  gc_DbmTranslation_fr_Text2200 : WSTRING(29) := "Activate Measuring Mast (A21)";
  gc_DbmTranslation_fr_Text2201 : WSTRING(76) := "Button for the calibration of min position mast measure encodeur  is pressed";
  gc_DbmTranslation_fr_Text2202 : WSTRING(76) := "Button for the calibration of max position mast measure encodeur  is pressed";
  gc_DbmTranslation_fr_Text2203 : WSTRING(58) := "Button for save min and max value of encodeur mast measure";
  gc_DbmTranslation_fr_Text2204 : WSTRING(60) := "Raz distance translation traveled with mast measure unfolded";
  gc_DbmTranslation_fr_Text2205 : WSTRING(13) := "Serial Number";
  gc_DbmTranslation_fr_Text2206 : WSTRING(18) := "BP Basket Validate";
  gc_DbmTranslation_fr_Text2207 : WSTRING(19) := "Key Filter Overload";
  gc_DbmTranslation_fr_Text2208 : WSTRING(13) := "Key Next Mode";
  gc_DbmTranslation_fr_Text2209 : WSTRING(13) := "Key Prev Mode";
  gc_DbmTranslation_fr_Text2210 : WSTRING(17) := "Key Signal Danger";
  gc_DbmTranslation_fr_Text2211 : WSTRING(18) := "Key Flash Light ON";
  gc_DbmTranslation_fr_Text2212 : WSTRING(18) := "Key Calib Mast Min";
  gc_DbmTranslation_fr_Text2213 : WSTRING(18) := "Key Calib Mast Max";
  gc_DbmTranslation_fr_Text2214 : WSTRING(17) := "KeyCalibMastValid";
  gc_DbmTranslation_fr_Text2215 : WSTRING(24) := "Key Generator Activation";
  gc_DbmTranslation_fr_Text2216 : WSTRING(31) := "Bypass pressure threshold alarm";
  gc_DbmTranslation_fr_Text2217 : WSTRING(66) := "DM_TELESCOPE_SENSOR_FAULT - Telescope In torlerance with inductive";
  gc_DbmTranslation_fr_Text2218 : WSTRING(78) := "DM_TELESCOPE_SENSOR_FAULT - Telescope torlerance when no movement is solicited";
  gc_DbmTranslation_fr_Text2219 : WSTRING(68) := "DM_TELESCOPE_SENSOR_FAULT - Telescope torlerance beetween 2 Channels";
  gc_DbmTranslation_fr_Text2220 : WSTRING(64) := "DM__INC_ALTERNATOR_CHARGE_FAULT - max treshold alternator regime";
  gc_DbmTranslation_fr_Text2221 : WSTRING(62) := "DM__INC_ALTERNATOR_CHARGE_FAULT - min treshold battery voltage";
  gc_DbmTranslation_fr_Text2222 : WSTRING(108) := "DM_C1_OUT_OF_RANGE_JOY_DELTA_ARM_48XS - min alarm value of joytick delta arm in % according batterie voltage";
  gc_DbmTranslation_fr_Text2223 : WSTRING(108) := "DM_C1_OUT_OF_RANGE_JOY_DELTA_ARM_48XS - max alarm value of joytick delta arm in % according batterie voltage";
  gc_DbmTranslation_fr_Text2224 : WSTRING(108) := "DM_C1_OUT_OF_RANGE_JOY_ARROW_ARM_48XS - min alarm value of joytick arrow arm in % according batterie voltage";
  gc_DbmTranslation_fr_Text2225 : WSTRING(108) := "DM_C1_OUT_OF_RANGE_JOY_ARROW_ARM_48XS - max alarm value of joytick arrow arm in % according batterie voltage";
  gc_DbmTranslation_fr_Text2226 : WSTRING(116) := "DM_C1_OUT_OF_RANGE_JOY_TELESCOPE_ARM_48XS - min alarm value of joytick telescope arm in % according batterie voltage";
  gc_DbmTranslation_fr_Text2227 : WSTRING(116) := "DM_C1_OUT_OF_RANGE_JOY_TELESCOPE_ARM_48XS - max alarm value of joytick telescope arm in % according batterie voltage";
  gc_DbmTranslation_fr_Text2228 : WSTRING(123) := "DM_C1_OUT_OF_RANGE_JOY_ROT_TURRET_ARM_48XS - min alarm value of joytick rotation turret arm in % according batterie voltage";
  gc_DbmTranslation_fr_Text2229 : WSTRING(123) := "DM_C1_OUT_OF_RANGE_JOY_ROT_TURRET_ARM_48XS - max alarm value of joytick rotation turret arm in % according batterie voltage";
  gc_DbmTranslation_fr_Text2230 : WSTRING(120) := "DM_C1_OUT_OF_RANGE_JOY_ADVANCEMENT_48XS - min alarm value of joytick rotation turret arm in % according batterie voltage";
  gc_DbmTranslation_fr_Text2231 : WSTRING(120) := "DM_C1_OUT_OF_RANGE_JOY_ADVANCEMENT_48XS - max alarm value of joytick rotation turret arm in % according batterie voltage";
  gc_DbmTranslation_fr_Text2232 : WSTRING(17) := "Time Bypass Fault";
  gc_DbmTranslation_fr_Text2233 : WSTRING(26) := "Timer for the Bypass fault";
  gc_DbmTranslation_fr_Text2234 : WSTRING(42) := "Inconsistency Nc No logical frame rotation";
  gc_DbmTranslation_fr_Text2235 : WSTRING(65) := "internal error , inconsistency between two channels and can error";
  gc_DbmTranslation_fr_Text2236 : WSTRING(37) := "Fault of Ev park brake axle osccilant";
  gc_DbmTranslation_fr_Text2237 : WSTRING(32) := "Fault of Ev park brake axle fixe";
  gc_DbmTranslation_fr_Text2238 : WSTRING(40) := "Fault of Ev service brake axle osccilant";
  gc_DbmTranslation_fr_Text2239 : WSTRING(35) := "Fault of Ev service brake axle fixe";
  gc_DbmTranslation_fr_Text2240 : WSTRING(30) := "Fault of Ev serice brake track";
  gc_DbmTranslation_fr_Text2241 : WSTRING(27) := "RM com can radio loss by C0";
  gc_DbmTranslation_fr_Text2242 : WSTRING(33) := "Ev 2nd Park Brake Axle Fixe Fault";
  gc_DbmTranslation_fr_Text2243 : WSTRING(33) := "Ev 2nd Park Brake Axle Osci Fault";
  gc_DbmTranslation_fr_Text2244 : WSTRING(0) := "";
  gc_DbmTranslation_fr_Text2245 : WSTRING(0) := "";
  gc_DbmTranslation_fr_Text2246 : WSTRING(0) := "";
  gc_DbmTranslation_fr_Text2247 : WSTRING(0) := "";
  gc_DbmTranslation_fr_Text2248 : WSTRING(0) := "";
  gc_DbmTranslation_fr_Text2249 : WSTRING(0) := "";
  gc_DbmTranslation_fr_Text2250 : WSTRING(0) := "";
  gc_DbmTranslation_fr_Text2251 : WSTRING(0) := "";
  gc_DbmTranslation_fr_Text2252 : WSTRING(0) := "";
  gc_DbmTranslation_fr_Text2253 : WSTRING(0) := "";
  gc_DbmTranslation_fr_Text2254 : WSTRING(0) := "";
  gc_DbmTranslation_fr_Text2255 : WSTRING(0) := "";
  gc_DbmTranslation_fr_Text2256 : WSTRING(0) := "";
  gc_DbmTranslation_fr_Text2257 : WSTRING(28) := "Additionnal Performance Func";
  gc_DbmTranslation_fr_Text2258 : WSTRING(21) := "Slope Case Less 2 Deg";
  gc_DbmTranslation_fr_Text2259 : WSTRING(21) := "Slope Case Less 4 Deg";
  gc_DbmTranslation_fr_Text2260 : WSTRING(21) := "Slope Case Less 6 Deg";
  gc_DbmTranslation_fr_Text2261 : WSTRING(23) := "Slope Case Higher 6 Deg";
  gc_DbmTranslation_fr_Text2262 : WSTRING(26) := "Turret In Speed Zone 2 Deg";
  gc_DbmTranslation_fr_Text2263 : WSTRING(26) := "Turret In Speed Zone 4 Deg";
  gc_DbmTranslation_fr_Text2264 : WSTRING(37) := "Turret In Speed Zone 2 Deg For Basket";
  gc_DbmTranslation_fr_Text2265 : WSTRING(21) := "Selected control post";
  gc_DbmTranslation_fr_Text2266 : WSTRING(23) := "Mast sensor position UP";
  gc_DbmTranslation_fr_Text2267 : WSTRING(40) := "Hydraulic valve uin down position sensor";
  gc_DbmTranslation_fr_Text2268 : WSTRING(28) := "Measuring mast sensor folded";
  gc_DbmTranslation_fr_Text2269 : WSTRING(35) := "Presence of sensor plate on machine";
  gc_DbmTranslation_fr_Text2270 : WSTRING(51) := "Recovery reduction ratio for the battery protection";
  gc_DbmTranslation_fr_Text2271 : WSTRING(21) := "Variable debug Neotec";
  gc_DbmTranslation_fr_Text2272 : WSTRING(21) := "Variable debug Neotec";
  gc_DbmTranslation_fr_Text2273 : WSTRING(21) := "Variable debug Neotec";
  gc_DbmTranslation_fr_Text2274 : WSTRING(21) := "Variable debug Neotec";
  gc_DbmTranslation_fr_Text2275 : WSTRING(21) := "Variable debug Neotec";
  gc_DbmTranslation_fr_Text2276 : WSTRING(21) := "Variable debug Neotec";
  gc_DbmTranslation_fr_Text2277 : WSTRING(21) := "Variable debug Neotec";
  gc_DbmTranslation_fr_Text2278 : WSTRING(21) := "Variable debug Neotec";
  gc_DbmTranslation_fr_Text2279 : WSTRING(21) := "Variable debug Neotec";
  gc_DbmTranslation_fr_Text2280 : WSTRING(21) := "Variable debug Neotec";
  gc_DbmTranslation_fr_Text2281 : WSTRING(21) := "Variable debug Neotec";
  gc_DbmTranslation_fr_Text2282 : WSTRING(21) := "Variable debug Neotec";
  gc_DbmTranslation_fr_Text2283 : WSTRING(21) := "Variable debug Neotec";
  gc_DbmTranslation_fr_Text2284 : WSTRING(21) := "Variable debug Neotec";
  gc_DbmTranslation_fr_Text2285 : WSTRING(21) := "Variable debug Neotec";
  gc_DbmTranslation_fr_Text2286 : WSTRING(21) := "Variable debug Neotec";
  gc_DbmTranslation_fr_Text2287 : WSTRING(21) := "Variable debug Neotec";
  gc_DbmTranslation_fr_Text2288 : WSTRING(21) := "Variable debug Neotec";
  gc_DbmTranslation_fr_Text2289 : WSTRING(21) := "Variable debug Neotec";
  gc_DbmTranslation_fr_Text2290 : WSTRING(21) := "Variable debug Neotec";
  gc_DbmTranslation_fr_Text2291 : WSTRING(21) := "Variable debug Neotec";
  gc_DbmTranslation_fr_Text2292 : WSTRING(21) := "Variable debug Neotec";
  gc_DbmTranslation_fr_Text2293 : WSTRING(21) := "Variable debug Neotec";
  gc_DbmTranslation_fr_Text2294 : WSTRING(21) := "Variable debug Neotec";
  gc_DbmTranslation_fr_Text2295 : WSTRING(21) := "Variable debug Neotec";
  gc_DbmTranslation_fr_Text2296 : WSTRING(21) := "Variable debug Neotec";
  gc_DbmTranslation_fr_Text2297 : WSTRING(21) := "Variable debug Neotec";
  gc_DbmTranslation_fr_Text2298 : WSTRING(21) := "Variable debug Neotec";
  gc_DbmTranslation_fr_Text2299 : WSTRING(21) := "Variable debug Neotec";
  gc_DbmTranslation_fr_Text2300 : WSTRING(21) := "Variable debug Neotec";
  gc_DbmTranslation_fr_Text2301 : WSTRING(21) := "Variable debug Neotec";
  gc_DbmTranslation_fr_Text2302 : WSTRING(21) := "Variable debug Neotec";
  gc_DbmTranslation_fr_Text2303 : WSTRING(21) := "Variable debug Neotec";
  gc_DbmTranslation_fr_Text2304 : WSTRING(21) := "Variable debug Neotec";
  gc_DbmTranslation_fr_Text2305 : WSTRING(21) := "Variable debug Neotec";
  gc_DbmTranslation_fr_Text2306 : WSTRING(21) := "Variable debug Neotec";
  gc_DbmTranslation_fr_Text2307 : WSTRING(21) := "Variable debug Neotec";
  gc_DbmTranslation_fr_Text2308 : WSTRING(21) := "Variable debug Neotec";
  gc_DbmTranslation_fr_Text2309 : WSTRING(21) := "Variable debug Neotec";
  gc_DbmTranslation_fr_Text2310 : WSTRING(21) := "Variable debug Neotec";
  gc_DbmTranslation_fr_Text2311 : WSTRING(64) := "Mesure de la température du liquide de refroidissement du moteur";
  gc_DbmTranslation_fr_Text2312 : WSTRING(58) := "Pression mesuré dans le système de lubrification du moteur";
  gc_DbmTranslation_fr_Text2313 : WSTRING(34) := "Vitesse actuelle du moteur calculé";
  gc_DbmTranslation_fr_Text2314 : WSTRING(56) := "Courant de l'alternateur principale du moteur thermique ";
  gc_DbmTranslation_fr_Text2315 : WSTRING(56) := "Etat du moteur : Motor stop, pre-start, Wram-Up,Starting";
  gc_DbmTranslation_fr_Text2316 : WSTRING(40) := "Tension mesuré aux bornes de la batterie";
  gc_DbmTranslation_fr_Text2317 : WSTRING(33) := "Commande de la vietesse du moteur";
  gc_DbmTranslation_fr_Text2318 : WSTRING(30) := "Override Control Mode (SPN695)";
  gc_DbmTranslation_fr_Text2319 : WSTRING(18) := "High pressure Oil ";
  gc_DbmTranslation_fr_Text2320 : WSTRING(14) := "Warmin gActive";
  gc_DbmTranslation_fr_Text2321 : WSTRING(10) := "Stop Motor";
  gc_DbmTranslation_fr_Text2322 : WSTRING(27) := "Regeneration SOC at maximum";
  gc_DbmTranslation_fr_Text2323 : WSTRING(61) := "Threshold maximum to autorize regeneration (Threshold of SOC)";
  gc_DbmTranslation_fr_Text2324 : WSTRING(42) := "Hysteresis for regeneration of SOC maximum";
  gc_DbmTranslation_fr_Text2325 : WSTRING(57) := "Number of time to refuse reloading from generator (Alarm)";
  gc_DbmTranslation_fr_Text2326 : WSTRING(61) := "Number of time to refuse reloading from generator (forbidden)";
  gc_DbmTranslation_fr_Text2327 : WSTRING(23) := "RPM motor maximum value";
  gc_DbmTranslation_fr_Text2328 : WSTRING(23) := "RPM motor minimum value";
  gc_DbmTranslation_fr_Text2329 : WSTRING(27) := "RPM for a movement with PVG";
  gc_DbmTranslation_fr_Text2330 : WSTRING(27) := "RPM for a movement with TOR";
  gc_DbmTranslation_fr_Text2331 : WSTRING(30) := "Hydraulic oil cold temperature";
  gc_DbmTranslation_fr_Text2332 : WSTRING(42) := "Capacity of the battery in ampere per hour";
  gc_DbmTranslation_fr_Text2333 : WSTRING(53) := "Number of element for the remaining regeneration time";
  gc_DbmTranslation_fr_Text2334 : WSTRING(61) := "Number of times the alarm regeneration threshold was exceeded";
  gc_DbmTranslation_fr_Text2335 : WSTRING(89) := "Number of times we exceeded the threshold of regeneration forbidden of the electric motor";
  gc_DbmTranslation_fr_Text2336 : WSTRING(25) := "Cold Oil Tank Temperature";
  gc_DbmTranslation_fr_Text2337 : WSTRING(30) := "Rpm Movements on Electric Mode";
  gc_DbmTranslation_fr_Text2338 : WSTRING(37) := "Rpm Translation on Rail Electric Mode";
  gc_DbmTranslation_fr_Text2339 : WSTRING(24) := "Rpm Oil Tank Temperature";
  gc_DbmTranslation_fr_Text2340 : WSTRING(18) := "Rpm Electric motor";
  gc_DbmTranslation_fr_Text2341 : WSTRING(12) := "Generator ON";
  gc_DbmTranslation_fr_Text2342 : WSTRING(23) := "Automatic mode activate";
  gc_DbmTranslation_fr_Text2343 : WSTRING(21) := "Silence mode activate";
  gc_DbmTranslation_fr_Text2344 : WSTRING(21) := "Forcing mode activate";
  gc_DbmTranslation_fr_Text2345 : WSTRING(24) := "Forcing regeneration Low";
  gc_DbmTranslation_fr_Text2346 : WSTRING(25) := "Forcing regeneration High";
  gc_DbmTranslation_fr_Text2347 : WSTRING(35) := "Remaining Regeneration time average";
  gc_DbmTranslation_fr_Text2348 : WSTRING(25) := "Ask Reload With Generator";
  gc_DbmTranslation_fr_Text2349 : WSTRING(27) := "Reloading With Generator On";
  gc_DbmTranslation_fr_Text2350 : WSTRING(24) := "Stop regeneration by SOC";
  gc_DbmTranslation_fr_Text2351 : WSTRING(24) := "Total regeneration Hours";
  gc_DbmTranslation_fr_Text2352 : WSTRING(31) := "Picto Cold Oil Tank Temperature";
  gc_DbmTranslation_fr_Text2353 : WSTRING(20) := "Total electric hours";
  gc_DbmTranslation_fr_Text2354 : WSTRING(37) := "Picto recovery reduction ratio active";
  gc_DbVarGrpNameTranslation_fr_Text2355 : WSTRING(17) := "NV_PARAMERTERS_C0";
  gc_DbVarGrpNameTranslation_fr_Text2356 : WSTRING(23) := "NV_PARAM_SPEED_MAX_RAIL";
  gc_DbVarGrpNameTranslation_fr_Text2357 : WSTRING(19) := "NV_PARAM_BRAKE_TEST";
  gc_DbVarGrpNameTranslation_fr_Text2358 : WSTRING(28) := "NV_PARAM_RAIL_WORK_SAFETY_C0";
  gc_DbVarGrpNameTranslation_fr_Text2359 : WSTRING(25) := "NV_PARAM_TRANSPORT_POS_C0";
  gc_DbVarGrpNameTranslation_fr_Text2360 : WSTRING(28) := "NV_PARAM_SELECT_CONTROL_POST";
  gc_DbVarGrpNameTranslation_fr_Text2361 : WSTRING(17) := "NV_PARAM_ALARM_C0";
  gc_DbVarGrpNameTranslation_fr_Text2362 : WSTRING(21) := "NV_PARAM_MAST_DISPLAY";
  gc_DbVarGrpNameTranslation_fr_Text2363 : WSTRING(17) := "NV_PARAMERTERS_C1";
  gc_DbVarGrpNameTranslation_fr_Text2364 : WSTRING(17) := "NV_PARAMERTERS_C1";
  gc_DbVarGrpNameTranslation_fr_Text2365 : WSTRING(17) := "NV_PARAM_MOTOR_C1";
  gc_DbVarGrpNameTranslation_fr_Text2366 : WSTRING(31) := "NV_PARAM_LIMIT_WORK_ENVELOPE_C1";
  gc_DbVarGrpNameTranslation_fr_Text2367 : WSTRING(24) := "NV_PARAM_MVT_END_STOP_C1";
  gc_DbVarGrpNameTranslation_fr_Text2368 : WSTRING(21) := "NV_PARAM_AUTO_STOP_C1";
  gc_DbVarGrpNameTranslation_fr_Text2369 : WSTRING(17) := "NV_PARAM_ALARM_C1";
  gc_DbVarGrpNameTranslation_fr_Text2370 : WSTRING(12) := "NV_OPTION_C0";
  gc_DbVarGrpNameTranslation_fr_Text2371 : WSTRING(12) := "NV_OPTION_C1";
  gc_DbmTranslation_fr_Texts : ARRAY[0..2371] OF POINTER TO WSTRING(123) := [ADR(gc_DbmTranslation_fr_Text0), ADR(gc_DbmTranslation_fr_Text1), ADR(gc_DbmTranslation_fr_Text2), ADR(gc_DbmTranslation_fr_Text3), ADR(gc_DbmTranslation_fr_Text4), ADR(gc_DbmTranslation_fr_Text5), ADR(gc_DbmTranslation_fr_Text6), ADR(gc_DbmTranslation_fr_Text7), ADR(gc_DbmTranslation_fr_Text8), ADR(gc_DbmTranslation_fr_Text9), ADR(gc_DbmTranslation_fr_Text10), ADR(gc_DbmTranslation_fr_Text11), ADR(gc_DbmTranslation_fr_Text12), ADR(gc_DbmTranslation_fr_Text13), ADR(gc_DbmTranslation_fr_Text14), ADR(gc_DbmTranslation_fr_Text15), ADR(gc_DbmTranslation_fr_Text16), ADR(gc_DbmTranslation_fr_Text17), ADR(gc_DbmTranslation_fr_Text18), ADR(gc_DbmTranslation_fr_Text19), ADR(gc_DbmTranslation_fr_Text20), ADR(gc_DbmTranslation_fr_Text21), ADR(gc_DbmTranslation_fr_Text22), ADR(gc_DbmTranslation_fr_Text23), ADR(gc_DbmTranslation_fr_Text24), ADR(gc_DbmTranslation_fr_Text25), ADR(gc_DbmTranslation_fr_Text26), ADR(gc_DbmTranslation_fr_Text27), ADR(gc_DbmTranslation_fr_Text28), ADR(gc_DbmTranslation_fr_Text29), ADR(gc_DbmTranslation_fr_Text30), ADR(gc_DbmTranslation_fr_Text31), ADR(gc_DbmTranslation_fr_Text32), ADR(gc_DbmTranslation_fr_Text33), ADR(gc_DbmTranslation_fr_Text34), ADR(gc_DbmTranslation_fr_Text35), ADR(gc_DbmTranslation_fr_Text36), ADR(gc_DbmTranslation_fr_Text37), ADR(gc_DbmTranslation_fr_Text38), ADR(gc_DbmTranslation_fr_Text39), ADR(gc_DbmTranslation_fr_Text40), ADR(gc_DbmTranslation_fr_Text41), ADR(gc_DbmTranslation_fr_Text42), ADR(gc_DbmTranslation_fr_Text43), ADR(gc_DbmTranslation_fr_Text44), ADR(gc_DbmTranslation_fr_Text45), ADR(gc_DbmTranslation_fr_Text46), ADR(gc_DbmTranslation_fr_Text47), ADR(gc_DbmTranslation_fr_Text48), ADR(gc_DbmTranslation_fr_Text49), ADR(gc_DbmTranslation_fr_Text50), ADR(gc_DbmTranslation_fr_Text51), ADR(gc_DbmTranslation_fr_Text52), ADR(gc_DbmTranslation_fr_Text53), ADR(gc_DbmTranslation_fr_Text54), ADR(gc_DbmTranslation_fr_Text55), ADR(gc_DbmTranslation_fr_Text56), ADR(gc_DbmTranslation_fr_Text57), ADR(gc_DbmTranslation_fr_Text58), ADR(gc_DbmTranslation_fr_Text59), ADR(gc_DbmTranslation_fr_Text60), ADR(gc_DbmTranslation_fr_Text61), ADR(gc_DbmTranslation_fr_Text62), ADR(gc_DbmTranslation_fr_Text63), ADR(gc_DbmTranslation_fr_Text64), ADR(gc_DbmTranslation_fr_Text65), ADR(gc_DbmTranslation_fr_Text66), ADR(gc_DbmTranslation_fr_Text67), ADR(gc_DbmTranslation_fr_Text68), ADR(gc_DbmTranslation_fr_Text69), ADR(gc_DbmTranslation_fr_Text70), ADR(gc_DbmTranslation_fr_Text71), ADR(gc_DbmTranslation_fr_Text72), ADR(gc_DbmTranslation_fr_Text73), ADR(gc_DbmTranslation_fr_Text74), ADR(gc_DbmTranslation_fr_Text75), ADR(gc_DbmTranslation_fr_Text76), ADR(gc_DbmTranslation_fr_Text77), ADR(gc_DbmTranslation_fr_Text78), ADR(gc_DbmTranslation_fr_Text79), ADR(gc_DbmTranslation_fr_Text80), ADR(gc_DbmTranslation_fr_Text81), ADR(gc_DbmTranslation_fr_Text82), ADR(gc_DbmTranslation_fr_Text83), ADR(gc_DbmTranslation_fr_Text84), ADR(gc_DbmTranslation_fr_Text85), ADR(gc_DbmTranslation_fr_Text86), ADR(gc_DbmTranslation_fr_Text87), ADR(gc_DbmTranslation_fr_Text88), ADR(gc_DbmTranslation_fr_Text89), ADR(gc_DbmTranslation_fr_Text90), ADR(gc_DbmTranslation_fr_Text91), ADR(gc_DbmTranslation_fr_Text92), ADR(gc_DbmTranslation_fr_Text93), ADR(gc_DbmTranslation_fr_Text94), ADR(gc_DbmTranslation_fr_Text95), ADR(gc_DbmTranslation_fr_Text96), ADR(gc_DbmTranslation_fr_Text97), ADR(gc_DbmTranslation_fr_Text98), ADR(gc_DbmTranslation_fr_Text99), ADR(gc_DbmTranslation_fr_Text100), ADR(gc_DbmTranslation_fr_Text101), ADR(gc_DbmTranslation_fr_Text102), ADR(gc_DbmTranslation_fr_Text103), ADR(gc_DbmTranslation_fr_Text104), ADR(gc_DbmTranslation_fr_Text105), ADR(gc_DbmTranslation_fr_Text106), ADR(gc_DbmTranslation_fr_Text107), ADR(gc_DbmTranslation_fr_Text108), ADR(gc_DbmTranslation_fr_Text109), ADR(gc_DbmTranslation_fr_Text110), ADR(gc_DbmTranslation_fr_Text111), ADR(gc_DbmTranslation_fr_Text112), ADR(gc_DbmTranslation_fr_Text113), ADR(gc_DbmTranslation_fr_Text114), ADR(gc_DbmTranslation_fr_Text115), ADR(gc_DbmTranslation_fr_Text116), ADR(gc_DbmTranslation_fr_Text117), ADR(gc_DbmTranslation_fr_Text118), ADR(gc_DbmTranslation_fr_Text119), ADR(gc_DbmTranslation_fr_Text120), ADR(gc_DbmTranslation_fr_Text121), ADR(gc_DbmTranslation_fr_Text122), ADR(gc_DbmTranslation_fr_Text123), ADR(gc_DbmTranslation_fr_Text124), ADR(gc_DbmTranslation_fr_Text125), ADR(gc_DbmTranslation_fr_Text126), ADR(gc_DbmTranslation_fr_Text127), ADR(gc_DbmTranslation_fr_Text128), ADR(gc_DbmTranslation_fr_Text129), ADR(gc_DbmTranslation_fr_Text130), ADR(gc_DbmTranslation_fr_Text131), ADR(gc_DbmTranslation_fr_Text132), ADR(gc_DbmTranslation_fr_Text133), ADR(gc_DbmTranslation_fr_Text134), ADR(gc_DbmTranslation_fr_Text135), ADR(gc_DbmTranslation_fr_Text136), ADR(gc_DbmTranslation_fr_Text137), ADR(gc_DbmTranslation_fr_Text138), ADR(gc_DbmTranslation_fr_Text139), ADR(gc_DbmTranslation_fr_Text140), ADR(gc_DbmTranslation_fr_Text141), ADR(gc_DbmTranslation_fr_Text142), ADR(gc_DbmTranslation_fr_Text143), ADR(gc_DbmTranslation_fr_Text144), ADR(gc_DbmTranslation_fr_Text145), ADR(gc_DbmTranslation_fr_Text146), ADR(gc_DbmTranslation_fr_Text147), ADR(gc_DbmTranslation_fr_Text148), ADR(gc_DbmTranslation_fr_Text149), ADR(gc_DbmTranslation_fr_Text150), ADR(gc_DbmTranslation_fr_Text151), ADR(gc_DbmTranslation_fr_Text152), ADR(gc_DbmTranslation_fr_Text153), ADR(gc_DbmTranslation_fr_Text154), ADR(gc_DbmTranslation_fr_Text155), ADR(gc_DbmTranslation_fr_Text156), ADR(gc_DbmTranslation_fr_Text157), ADR(gc_DbmTranslation_fr_Text158), ADR(gc_DbmTranslation_fr_Text159), ADR(gc_DbmTranslation_fr_Text160), ADR(gc_DbmTranslation_fr_Text161), ADR(gc_DbmTranslation_fr_Text162), ADR(gc_DbmTranslation_fr_Text163), ADR(gc_DbmTranslation_fr_Text164), ADR(gc_DbmTranslation_fr_Text165), ADR(gc_DbmTranslation_fr_Text166), ADR(gc_DbmTranslation_fr_Text167), ADR(gc_DbmTranslation_fr_Text168), ADR(gc_DbmTranslation_fr_Text169), ADR(gc_DbmTranslation_fr_Text170), ADR(gc_DbmTranslation_fr_Text171), ADR(gc_DbmTranslation_fr_Text172), ADR(gc_DbmTranslation_fr_Text173), ADR(gc_DbmTranslation_fr_Text174), ADR(gc_DbmTranslation_fr_Text175), ADR(gc_DbmTranslation_fr_Text176), ADR(gc_DbmTranslation_fr_Text177), ADR(gc_DbmTranslation_fr_Text178), ADR(gc_DbmTranslation_fr_Text179), ADR(gc_DbmTranslation_fr_Text180), ADR(gc_DbmTranslation_fr_Text181), ADR(gc_DbmTranslation_fr_Text182), ADR(gc_DbmTranslation_fr_Text183), ADR(gc_DbmTranslation_fr_Text184), ADR(gc_DbmTranslation_fr_Text185), ADR(gc_DbmTranslation_fr_Text186), ADR(gc_DbmTranslation_fr_Text187), ADR(gc_DbmTranslation_fr_Text188), ADR(gc_DbmTranslation_fr_Text189), ADR(gc_DbmTranslation_fr_Text190), ADR(gc_DbmTranslation_fr_Text191), ADR(gc_DbmTranslation_fr_Text192), ADR(gc_DbmTranslation_fr_Text193), ADR(gc_DbmTranslation_fr_Text194), ADR(gc_DbmTranslation_fr_Text195), ADR(gc_DbmTranslation_fr_Text196), ADR(gc_DbmTranslation_fr_Text197), ADR(gc_DbmTranslation_fr_Text198), ADR(gc_DbmTranslation_fr_Text199), ADR(gc_DbmTranslation_fr_Text200), ADR(gc_DbmTranslation_fr_Text201), ADR(gc_DbmTranslation_fr_Text202), ADR(gc_DbmTranslation_fr_Text203), ADR(gc_DbmTranslation_fr_Text204), ADR(gc_DbmTranslation_fr_Text205), ADR(gc_DbmTranslation_fr_Text206), ADR(gc_DbmTranslation_fr_Text207), ADR(gc_DbmTranslation_fr_Text208), ADR(gc_DbmTranslation_fr_Text209), ADR(gc_DbmTranslation_fr_Text210), ADR(gc_DbmTranslation_fr_Text211), ADR(gc_DbmTranslation_fr_Text212), ADR(gc_DbmTranslation_fr_Text213), ADR(gc_DbmTranslation_fr_Text214), ADR(gc_DbmTranslation_fr_Text215), ADR(gc_DbmTranslation_fr_Text216), ADR(gc_DbmTranslation_fr_Text217), ADR(gc_DbmTranslation_fr_Text218), ADR(gc_DbmTranslation_fr_Text219), ADR(gc_DbmTranslation_fr_Text220), ADR(gc_DbmTranslation_fr_Text221), ADR(gc_DbmTranslation_fr_Text222), ADR(gc_DbmTranslation_fr_Text223), ADR(gc_DbmTranslation_fr_Text224), ADR(gc_DbmTranslation_fr_Text225), ADR(gc_DbmTranslation_fr_Text226), ADR(gc_DbmTranslation_fr_Text227), ADR(gc_DbmTranslation_fr_Text228), ADR(gc_DbmTranslation_fr_Text229), ADR(gc_DbmTranslation_fr_Text230), ADR(gc_DbmTranslation_fr_Text231), ADR(gc_DbmTranslation_fr_Text232), ADR(gc_DbmTranslation_fr_Text233), ADR(gc_DbmTranslation_fr_Text234), ADR(gc_DbmTranslation_fr_Text235), ADR(gc_DbmTranslation_fr_Text236), ADR(gc_DbmTranslation_fr_Text237), ADR(gc_DbmTranslation_fr_Text238), ADR(gc_DbmTranslation_fr_Text239), ADR(gc_DbmTranslation_fr_Text240), ADR(gc_DbmTranslation_fr_Text241), ADR(gc_DbmTranslation_fr_Text242), ADR(gc_DbmTranslation_fr_Text243), ADR(gc_DbmTranslation_fr_Text244), ADR(gc_DbmTranslation_fr_Text245), ADR(gc_DbmTranslation_fr_Text246), ADR(gc_DbmTranslation_fr_Text247), ADR(gc_DbmTranslation_fr_Text248), ADR(gc_DbmTranslation_fr_Text249), ADR(gc_DbmTranslation_fr_Text250), ADR(gc_DbmTranslation_fr_Text251), ADR(gc_DbmTranslation_fr_Text252), ADR(gc_DbmTranslation_fr_Text253), ADR(gc_DbmTranslation_fr_Text254), ADR(gc_DbmTranslation_fr_Text255), ADR(gc_DbmTranslation_fr_Text256), ADR(gc_DbmTranslation_fr_Text257), ADR(gc_DbmTranslation_fr_Text258), ADR(gc_DbmTranslation_fr_Text259), ADR(gc_DbmTranslation_fr_Text260), ADR(gc_DbmTranslation_fr_Text261), ADR(gc_DbmTranslation_fr_Text262), ADR(gc_DbmTranslation_fr_Text263), ADR(gc_DbmTranslation_fr_Text264), ADR(gc_DbmTranslation_fr_Text265), ADR(gc_DbmTranslation_fr_Text266), ADR(gc_DbmTranslation_fr_Text267), ADR(gc_DbmTranslation_fr_Text268), ADR(gc_DbmTranslation_fr_Text269), ADR(gc_DbmTranslation_fr_Text270), ADR(gc_DbmTranslation_fr_Text271), ADR(gc_DbmTranslation_fr_Text272), ADR(gc_DbmTranslation_fr_Text273), ADR(gc_DbmTranslation_fr_Text274), ADR(gc_DbmTranslation_fr_Text275), ADR(gc_DbmTranslation_fr_Text276), ADR(gc_DbmTranslation_fr_Text277), ADR(gc_DbmTranslation_fr_Text278), ADR(gc_DbmTranslation_fr_Text279), ADR(gc_DbmTranslation_fr_Text280), ADR(gc_DbmTranslation_fr_Text281), ADR(gc_DbmTranslation_fr_Text282), ADR(gc_DbmTranslation_fr_Text283), ADR(gc_DbmTranslation_fr_Text284), ADR(gc_DbmTranslation_fr_Text285), ADR(gc_DbmTranslation_fr_Text286), ADR(gc_DbmTranslation_fr_Text287), ADR(gc_DbmTranslation_fr_Text288), ADR(gc_DbmTranslation_fr_Text289), ADR(gc_DbmTranslation_fr_Text290), ADR(gc_DbmTranslation_fr_Text291), ADR(gc_DbmTranslation_fr_Text292), ADR(gc_DbmTranslation_fr_Text293), ADR(gc_DbmTranslation_fr_Text294), ADR(gc_DbmTranslation_fr_Text295), ADR(gc_DbmTranslation_fr_Text296), ADR(gc_DbmTranslation_fr_Text297), ADR(gc_DbmTranslation_fr_Text298), ADR(gc_DbmTranslation_fr_Text299), ADR(gc_DbmTranslation_fr_Text300), ADR(gc_DbmTranslation_fr_Text301), ADR(gc_DbmTranslation_fr_Text302), ADR(gc_DbmTranslation_fr_Text303), ADR(gc_DbmTranslation_fr_Text304), ADR(gc_DbmTranslation_fr_Text305), ADR(gc_DbmTranslation_fr_Text306), ADR(gc_DbmTranslation_fr_Text307), ADR(gc_DbmTranslation_fr_Text308), ADR(gc_DbmTranslation_fr_Text309), ADR(gc_DbmTranslation_fr_Text310), ADR(gc_DbmTranslation_fr_Text311), ADR(gc_DbmTranslation_fr_Text312), ADR(gc_DbmTranslation_fr_Text313), ADR(gc_DbmTranslation_fr_Text314), ADR(gc_DbmTranslation_fr_Text315), ADR(gc_DbmTranslation_fr_Text316), ADR(gc_DbmTranslation_fr_Text317), ADR(gc_DbmTranslation_fr_Text318), ADR(gc_DbmTranslation_fr_Text319), ADR(gc_DbmTranslation_fr_Text320), ADR(gc_DbmTranslation_fr_Text321), ADR(gc_DbmTranslation_fr_Text322), ADR(gc_DbmTranslation_fr_Text323), ADR(gc_DbmTranslation_fr_Text324), ADR(gc_DbmTranslation_fr_Text325), ADR(gc_DbmTranslation_fr_Text326), ADR(gc_DbmTranslation_fr_Text327), ADR(gc_DbmTranslation_fr_Text328), ADR(gc_DbmTranslation_fr_Text329), ADR(gc_DbmTranslation_fr_Text330), ADR(gc_DbmTranslation_fr_Text331), ADR(gc_DbmTranslation_fr_Text332), ADR(gc_DbmTranslation_fr_Text333), ADR(gc_DbmTranslation_fr_Text334), ADR(gc_DbmTranslation_fr_Text335), ADR(gc_DbmTranslation_fr_Text336), ADR(gc_DbmTranslation_fr_Text337), ADR(gc_DbmTranslation_fr_Text338), ADR(gc_DbmTranslation_fr_Text339), ADR(gc_DbmTranslation_fr_Text340), ADR(gc_DbmTranslation_fr_Text341), ADR(gc_DbmTranslation_fr_Text342), ADR(gc_DbmTranslation_fr_Text343), ADR(gc_DbmTranslation_fr_Text344), ADR(gc_DbmTranslation_fr_Text345), ADR(gc_DbmTranslation_fr_Text346), ADR(gc_DbmTranslation_fr_Text347), ADR(gc_DbmTranslation_fr_Text348), ADR(gc_DbmTranslation_fr_Text349), ADR(gc_DbmTranslation_fr_Text350), ADR(gc_DbmTranslation_fr_Text351), ADR(gc_DbmTranslation_fr_Text352), ADR(gc_DbmTranslation_fr_Text353), ADR(gc_DbmTranslation_fr_Text354), ADR(gc_DbmTranslation_fr_Text355), ADR(gc_DbmTranslation_fr_Text356), ADR(gc_DbmTranslation_fr_Text357), ADR(gc_DbmTranslation_fr_Text358), ADR(gc_DbmTranslation_fr_Text359), ADR(gc_DbmTranslation_fr_Text360), ADR(gc_DbmTranslation_fr_Text361), ADR(gc_DbmTranslation_fr_Text362), ADR(gc_DbmTranslation_fr_Text363), ADR(gc_DbmTranslation_fr_Text364), ADR(gc_DbmTranslation_fr_Text365), ADR(gc_DbmTranslation_fr_Text366), ADR(gc_DbmTranslation_fr_Text367), ADR(gc_DbmTranslation_fr_Text368), ADR(gc_DbmTranslation_fr_Text369), ADR(gc_DbmTranslation_fr_Text370), ADR(gc_DbmTranslation_fr_Text371), ADR(gc_DbmTranslation_fr_Text372), ADR(gc_DbmTranslation_fr_Text373), ADR(gc_DbmTranslation_fr_Text374), ADR(gc_DbmTranslation_fr_Text375), ADR(gc_DbmTranslation_fr_Text376), ADR(gc_DbmTranslation_fr_Text377), ADR(gc_DbmTranslation_fr_Text378), ADR(gc_DbmTranslation_fr_Text379), ADR(gc_DbmTranslation_fr_Text380), ADR(gc_DbmTranslation_fr_Text381), ADR(gc_DbmTranslation_fr_Text382), ADR(gc_DbmTranslation_fr_Text383), ADR(gc_DbmTranslation_fr_Text384), ADR(gc_DbmTranslation_fr_Text385), ADR(gc_DbmTranslation_fr_Text386), ADR(gc_DbmTranslation_fr_Text387), ADR(gc_DbmTranslation_fr_Text388), ADR(gc_DbmTranslation_fr_Text389), ADR(gc_DbmTranslation_fr_Text390), ADR(gc_DbmTranslation_fr_Text391), ADR(gc_DbmTranslation_fr_Text392), ADR(gc_DbmTranslation_fr_Text393), ADR(gc_DbmTranslation_fr_Text394), ADR(gc_DbmTranslation_fr_Text395), ADR(gc_DbmTranslation_fr_Text396), ADR(gc_DbmTranslation_fr_Text397), ADR(gc_DbmTranslation_fr_Text398), ADR(gc_DbmTranslation_fr_Text399), ADR(gc_DbmTranslation_fr_Text400), ADR(gc_DbmTranslation_fr_Text401), ADR(gc_DbmTranslation_fr_Text402), ADR(gc_DbmTranslation_fr_Text403), ADR(gc_DbmTranslation_fr_Text404), ADR(gc_DbmTranslation_fr_Text405), ADR(gc_DbmTranslation_fr_Text406), ADR(gc_DbmTranslation_fr_Text407), ADR(gc_DbmTranslation_fr_Text408), ADR(gc_DbmTranslation_fr_Text409), ADR(gc_DbmTranslation_fr_Text410), ADR(gc_DbmTranslation_fr_Text411), ADR(gc_DbmTranslation_fr_Text412), ADR(gc_DbmTranslation_fr_Text413), ADR(gc_DbmTranslation_fr_Text414), ADR(gc_DbmTranslation_fr_Text415), ADR(gc_DbmTranslation_fr_Text416), ADR(gc_DbmTranslation_fr_Text417), ADR(gc_DbmTranslation_fr_Text418), ADR(gc_DbmTranslation_fr_Text419), ADR(gc_DbmTranslation_fr_Text420), ADR(gc_DbmTranslation_fr_Text421), ADR(gc_DbmTranslation_fr_Text422), ADR(gc_DbmTranslation_fr_Text423), ADR(gc_DbmTranslation_fr_Text424), ADR(gc_DbmTranslation_fr_Text425), ADR(gc_DbmTranslation_fr_Text426), ADR(gc_DbmTranslation_fr_Text427), ADR(gc_DbmTranslation_fr_Text428), ADR(gc_DbmTranslation_fr_Text429), ADR(gc_DbmTranslation_fr_Text430), ADR(gc_DbmTranslation_fr_Text431), ADR(gc_DbmTranslation_fr_Text432), ADR(gc_DbmTranslation_fr_Text433), ADR(gc_DbmTranslation_fr_Text434), ADR(gc_DbmTranslation_fr_Text435), ADR(gc_DbmTranslation_fr_Text436), ADR(gc_DbmTranslation_fr_Text437), ADR(gc_DbmTranslation_fr_Text438), ADR(gc_DbmTranslation_fr_Text439), ADR(gc_DbmTranslation_fr_Text440), ADR(gc_DbmTranslation_fr_Text441), ADR(gc_DbmTranslation_fr_Text442), ADR(gc_DbmTranslation_fr_Text443), ADR(gc_DbmTranslation_fr_Text444), ADR(gc_DbmTranslation_fr_Text445), ADR(gc_DbmTranslation_fr_Text446), ADR(gc_DbmTranslation_fr_Text447), ADR(gc_DbmTranslation_fr_Text448), ADR(gc_DbmTranslation_fr_Text449), ADR(gc_DbmTranslation_fr_Text450), ADR(gc_DbmTranslation_fr_Text451), ADR(gc_DbmTranslation_fr_Text452), ADR(gc_DbmTranslation_fr_Text453), ADR(gc_DbmTranslation_fr_Text454), ADR(gc_DbmTranslation_fr_Text455), ADR(gc_DbmTranslation_fr_Text456), ADR(gc_DbmTranslation_fr_Text457), ADR(gc_DbmTranslation_fr_Text458), ADR(gc_DbmTranslation_fr_Text459), ADR(gc_DbmTranslation_fr_Text460), ADR(gc_DbmTranslation_fr_Text461), ADR(gc_DbmTranslation_fr_Text462), ADR(gc_DbmTranslation_fr_Text463), ADR(gc_DbmTranslation_fr_Text464), ADR(gc_DbmTranslation_fr_Text465), ADR(gc_DbmTranslation_fr_Text466), ADR(gc_DbmTranslation_fr_Text467), ADR(gc_DbmTranslation_fr_Text468), ADR(gc_DbmTranslation_fr_Text469), ADR(gc_DbmTranslation_fr_Text470), ADR(gc_DbmTranslation_fr_Text471), ADR(gc_DbmTranslation_fr_Text472), ADR(gc_DbmTranslation_fr_Text473), ADR(gc_DbmTranslation_fr_Text474), ADR(gc_DbmTranslation_fr_Text475), ADR(gc_DbmTranslation_fr_Text476), ADR(gc_DbmTranslation_fr_Text477), ADR(gc_DbmTranslation_fr_Text478), ADR(gc_DbmTranslation_fr_Text479), ADR(gc_DbmTranslation_fr_Text480), ADR(gc_DbmTranslation_fr_Text481), ADR(gc_DbmTranslation_fr_Text482), ADR(gc_DbmTranslation_fr_Text483), ADR(gc_DbmTranslation_fr_Text484), ADR(gc_DbmTranslation_fr_Text485), ADR(gc_DbmTranslation_fr_Text486), ADR(gc_DbmTranslation_fr_Text487), ADR(gc_DbmTranslation_fr_Text488), ADR(gc_DbmTranslation_fr_Text489), ADR(gc_DbmTranslation_fr_Text490), ADR(gc_DbmTranslation_fr_Text491), ADR(gc_DbmTranslation_fr_Text492), ADR(gc_DbmTranslation_fr_Text493), ADR(gc_DbmTranslation_fr_Text494), ADR(gc_DbmTranslation_fr_Text495), ADR(gc_DbmTranslation_fr_Text496), ADR(gc_DbmTranslation_fr_Text497), ADR(gc_DbmTranslation_fr_Text498), ADR(gc_DbmTranslation_fr_Text499), ADR(gc_DbmTranslation_fr_Text500), ADR(gc_DbmTranslation_fr_Text501), ADR(gc_DbmTranslation_fr_Text502), ADR(gc_DbmTranslation_fr_Text503), ADR(gc_DbmTranslation_fr_Text504), ADR(gc_DbmTranslation_fr_Text505), ADR(gc_DbmTranslation_fr_Text506), ADR(gc_DbmTranslation_fr_Text507), ADR(gc_DbmTranslation_fr_Text508), ADR(gc_DbmTranslation_fr_Text509), ADR(gc_DbmTranslation_fr_Text510), ADR(gc_DbmTranslation_fr_Text511), ADR(gc_DbmTranslation_fr_Text512), ADR(gc_DbmTranslation_fr_Text513), ADR(gc_DbmTranslation_fr_Text514), ADR(gc_DbmTranslation_fr_Text515), ADR(gc_DbmTranslation_fr_Text516), ADR(gc_DbmTranslation_fr_Text517), ADR(gc_DbmTranslation_fr_Text518), ADR(gc_DbmTranslation_fr_Text519), ADR(gc_DbmTranslation_fr_Text520), ADR(gc_DbmTranslation_fr_Text521), ADR(gc_DbmTranslation_fr_Text522), ADR(gc_DbmTranslation_fr_Text523), ADR(gc_DbmTranslation_fr_Text524), ADR(gc_DbmTranslation_fr_Text525), ADR(gc_DbmTranslation_fr_Text526), ADR(gc_DbmTranslation_fr_Text527), ADR(gc_DbmTranslation_fr_Text528), ADR(gc_DbmTranslation_fr_Text529), ADR(gc_DbmTranslation_fr_Text530), ADR(gc_DbmTranslation_fr_Text531), ADR(gc_DbmTranslation_fr_Text532), ADR(gc_DbmTranslation_fr_Text533), ADR(gc_DbmTranslation_fr_Text534), ADR(gc_DbmTranslation_fr_Text535), ADR(gc_DbmTranslation_fr_Text536), ADR(gc_DbmTranslation_fr_Text537), ADR(gc_DbmTranslation_fr_Text538), ADR(gc_DbmTranslation_fr_Text539), ADR(gc_DbmTranslation_fr_Text540), ADR(gc_DbmTranslation_fr_Text541), ADR(gc_DbmTranslation_fr_Text542), ADR(gc_DbmTranslation_fr_Text543), ADR(gc_DbmTranslation_fr_Text544), ADR(gc_DbmTranslation_fr_Text545), ADR(gc_DbmTranslation_fr_Text546), ADR(gc_DbmTranslation_fr_Text547), ADR(gc_DbmTranslation_fr_Text548), ADR(gc_DbmTranslation_fr_Text549), ADR(gc_DbmTranslation_fr_Text550), ADR(gc_DbmTranslation_fr_Text551), ADR(gc_DbmTranslation_fr_Text552), ADR(gc_DbmTranslation_fr_Text553), ADR(gc_DbmTranslation_fr_Text554), ADR(gc_DbmTranslation_fr_Text555), ADR(gc_DbmTranslation_fr_Text556), ADR(gc_DbmTranslation_fr_Text557), ADR(gc_DbmTranslation_fr_Text558), ADR(gc_DbmTranslation_fr_Text559), ADR(gc_DbmTranslation_fr_Text560), ADR(gc_DbmTranslation_fr_Text561), ADR(gc_DbmTranslation_fr_Text562), ADR(gc_DbmTranslation_fr_Text563), ADR(gc_DbmTranslation_fr_Text564), ADR(gc_DbmTranslation_fr_Text565), ADR(gc_DbmTranslation_fr_Text566), ADR(gc_DbmTranslation_fr_Text567), ADR(gc_DbmTranslation_fr_Text568), ADR(gc_DbmTranslation_fr_Text569), ADR(gc_DbmTranslation_fr_Text570), ADR(gc_DbmTranslation_fr_Text571), ADR(gc_DbmTranslation_fr_Text572), ADR(gc_DbmTranslation_fr_Text573), ADR(gc_DbmTranslation_fr_Text574), ADR(gc_DbmTranslation_fr_Text575), ADR(gc_DbmTranslation_fr_Text576), ADR(gc_DbmTranslation_fr_Text577), ADR(gc_DbmTranslation_fr_Text578), ADR(gc_DbmTranslation_fr_Text579), ADR(gc_DbmTranslation_fr_Text580), ADR(gc_DbmTranslation_fr_Text581), ADR(gc_DbmTranslation_fr_Text582), ADR(gc_DbmTranslation_fr_Text583), ADR(gc_DbmTranslation_fr_Text584), ADR(gc_DbmTranslation_fr_Text585), ADR(gc_DbmTranslation_fr_Text586), ADR(gc_DbmTranslation_fr_Text587), ADR(gc_DbmTranslation_fr_Text588), ADR(gc_DbmTranslation_fr_Text589), ADR(gc_DbmTranslation_fr_Text590), ADR(gc_DbmTranslation_fr_Text591), ADR(gc_DbmTranslation_fr_Text592), ADR(gc_DbmTranslation_fr_Text593), ADR(gc_DbmTranslation_fr_Text594), ADR(gc_DbmTranslation_fr_Text595), ADR(gc_DbmTranslation_fr_Text596), ADR(gc_DbmTranslation_fr_Text597), ADR(gc_DbmTranslation_fr_Text598), ADR(gc_DbmTranslation_fr_Text599), ADR(gc_DbmTranslation_fr_Text600), ADR(gc_DbmTranslation_fr_Text601), ADR(gc_DbmTranslation_fr_Text602), ADR(gc_DbmTranslation_fr_Text603), ADR(gc_DbmTranslation_fr_Text604), ADR(gc_DbmTranslation_fr_Text605), ADR(gc_DbmTranslation_fr_Text606), ADR(gc_DbmTranslation_fr_Text607), ADR(gc_DbmTranslation_fr_Text608), ADR(gc_DbmTranslation_fr_Text609), ADR(gc_DbmTranslation_fr_Text610), ADR(gc_DbmTranslation_fr_Text611), ADR(gc_DbmTranslation_fr_Text612), ADR(gc_DbmTranslation_fr_Text613), ADR(gc_DbmTranslation_fr_Text614), ADR(gc_DbmTranslation_fr_Text615), ADR(gc_DbmTranslation_fr_Text616), ADR(gc_DbmTranslation_fr_Text617), ADR(gc_DbmTranslation_fr_Text618), ADR(gc_DbmTranslation_fr_Text619), ADR(gc_DbmTranslation_fr_Text620), ADR(gc_DbmTranslation_fr_Text621), ADR(gc_DbmTranslation_fr_Text622), ADR(gc_DbmTranslation_fr_Text623), ADR(gc_DbmTranslation_fr_Text624), ADR(gc_DbmTranslation_fr_Text625), ADR(gc_DbmTranslation_fr_Text626), ADR(gc_DbmTranslation_fr_Text627), ADR(gc_DbmTranslation_fr_Text628), ADR(gc_DbmTranslation_fr_Text629), ADR(gc_DbmTranslation_fr_Text630), ADR(gc_DbmTranslation_fr_Text631), ADR(gc_DbmTranslation_fr_Text632), ADR(gc_DbmTranslation_fr_Text633), ADR(gc_DbmTranslation_fr_Text634), ADR(gc_DbmTranslation_fr_Text635), ADR(gc_DbmTranslation_fr_Text636), ADR(gc_DbmTranslation_fr_Text637), ADR(gc_DbmTranslation_fr_Text638), ADR(gc_DbmTranslation_fr_Text639), ADR(gc_DbmTranslation_fr_Text640), ADR(gc_DbmTranslation_fr_Text641), ADR(gc_DbmTranslation_fr_Text642), ADR(gc_DbmTranslation_fr_Text643), ADR(gc_DbmTranslation_fr_Text644), ADR(gc_DbmTranslation_fr_Text645), ADR(gc_DbmTranslation_fr_Text646), ADR(gc_DbmTranslation_fr_Text647), ADR(gc_DbmTranslation_fr_Text648), ADR(gc_DbmTranslation_fr_Text649), ADR(gc_DbmTranslation_fr_Text650), ADR(gc_DbmTranslation_fr_Text651), ADR(gc_DbmTranslation_fr_Text652), ADR(gc_DbmTranslation_fr_Text653), ADR(gc_DbmTranslation_fr_Text654), ADR(gc_DbmTranslation_fr_Text655), ADR(gc_DbmTranslation_fr_Text656), ADR(gc_DbmTranslation_fr_Text657), ADR(gc_DbmTranslation_fr_Text658), ADR(gc_DbmTranslation_fr_Text659), ADR(gc_DbmTranslation_fr_Text660), ADR(gc_DbmTranslation_fr_Text661), ADR(gc_DbmTranslation_fr_Text662), ADR(gc_DbmTranslation_fr_Text663), ADR(gc_DbmTranslation_fr_Text664), ADR(gc_DbmTranslation_fr_Text665), ADR(gc_DbmTranslation_fr_Text666), ADR(gc_DbmTranslation_fr_Text667), ADR(gc_DbmTranslation_fr_Text668), ADR(gc_DbmTranslation_fr_Text669), ADR(gc_DbmTranslation_fr_Text670), ADR(gc_DbmTranslation_fr_Text671), ADR(gc_DbmTranslation_fr_Text672), ADR(gc_DbmTranslation_fr_Text673), ADR(gc_DbmTranslation_fr_Text674), ADR(gc_DbmTranslation_fr_Text675), ADR(gc_DbmTranslation_fr_Text676), ADR(gc_DbmTranslation_fr_Text677), ADR(gc_DbmTranslation_fr_Text678), ADR(gc_DbmTranslation_fr_Text679), ADR(gc_DbmTranslation_fr_Text680), ADR(gc_DbmTranslation_fr_Text681), ADR(gc_DbmTranslation_fr_Text682), ADR(gc_DbmTranslation_fr_Text683), ADR(gc_DbmTranslation_fr_Text684), ADR(gc_DbmTranslation_fr_Text685), ADR(gc_DbmTranslation_fr_Text686), ADR(gc_DbmTranslation_fr_Text687), ADR(gc_DbmTranslation_fr_Text688), ADR(gc_DbmTranslation_fr_Text689), ADR(gc_DbmTranslation_fr_Text690), ADR(gc_DbmTranslation_fr_Text691), ADR(gc_DbmTranslation_fr_Text692), ADR(gc_DbmTranslation_fr_Text693), ADR(gc_DbmTranslation_fr_Text694), ADR(gc_DbmTranslation_fr_Text695), ADR(gc_DbmTranslation_fr_Text696), ADR(gc_DbmTranslation_fr_Text697), ADR(gc_DbmTranslation_fr_Text698), ADR(gc_DbmTranslation_fr_Text699), ADR(gc_DbmTranslation_fr_Text700), ADR(gc_DbmTranslation_fr_Text701), ADR(gc_DbmTranslation_fr_Text702), ADR(gc_DbmTranslation_fr_Text703), ADR(gc_DbmTranslation_fr_Text704), ADR(gc_DbmTranslation_fr_Text705), ADR(gc_DbmTranslation_fr_Text706), ADR(gc_DbmTranslation_fr_Text707), ADR(gc_DbmTranslation_fr_Text708), ADR(gc_DbmTranslation_fr_Text709), ADR(gc_DbmTranslation_fr_Text710), ADR(gc_DbmTranslation_fr_Text711), ADR(gc_DbmTranslation_fr_Text712), ADR(gc_DbmTranslation_fr_Text713), ADR(gc_DbmTranslation_fr_Text714), ADR(gc_DbmTranslation_fr_Text715), ADR(gc_DbmTranslation_fr_Text716), ADR(gc_DbmTranslation_fr_Text717), ADR(gc_DbmTranslation_fr_Text718), ADR(gc_DbmTranslation_fr_Text719), ADR(gc_DbmTranslation_fr_Text720), ADR(gc_DbmTranslation_fr_Text721), ADR(gc_DbmTranslation_fr_Text722), ADR(gc_DbmTranslation_fr_Text723), ADR(gc_DbmTranslation_fr_Text724), ADR(gc_DbmTranslation_fr_Text725), ADR(gc_DbmTranslation_fr_Text726), ADR(gc_DbmTranslation_fr_Text727), ADR(gc_DbmTranslation_fr_Text728), ADR(gc_DbmTranslation_fr_Text729), ADR(gc_DbmTranslation_fr_Text730), ADR(gc_DbmTranslation_fr_Text731), ADR(gc_DbmTranslation_fr_Text732), ADR(gc_DbmTranslation_fr_Text733), ADR(gc_DbmTranslation_fr_Text734), ADR(gc_DbmTranslation_fr_Text735), ADR(gc_DbmTranslation_fr_Text736), ADR(gc_DbmTranslation_fr_Text737), ADR(gc_DbmTranslation_fr_Text738), ADR(gc_DbmTranslation_fr_Text739), ADR(gc_DbmTranslation_fr_Text740), ADR(gc_DbmTranslation_fr_Text741), ADR(gc_DbmTranslation_fr_Text742), ADR(gc_DbmTranslation_fr_Text743), ADR(gc_DbmTranslation_fr_Text744), ADR(gc_DbmTranslation_fr_Text745), ADR(gc_DbmTranslation_fr_Text746), ADR(gc_DbmTranslation_fr_Text747), ADR(gc_DbmTranslation_fr_Text748), ADR(gc_DbmTranslation_fr_Text749), ADR(gc_DbmTranslation_fr_Text750), ADR(gc_DbmTranslation_fr_Text751), ADR(gc_DbmTranslation_fr_Text752), ADR(gc_DbmTranslation_fr_Text753), ADR(gc_DbmTranslation_fr_Text754), ADR(gc_DbmTranslation_fr_Text755), ADR(gc_DbmTranslation_fr_Text756), ADR(gc_DbmTranslation_fr_Text757), ADR(gc_DbmTranslation_fr_Text758), ADR(gc_DbmTranslation_fr_Text759), ADR(gc_DbmTranslation_fr_Text760), ADR(gc_DbmTranslation_fr_Text761), ADR(gc_DbmTranslation_fr_Text762), ADR(gc_DbmTranslation_fr_Text763), ADR(gc_DbmTranslation_fr_Text764), ADR(gc_DbmTranslation_fr_Text765), ADR(gc_DbmTranslation_fr_Text766), ADR(gc_DbmTranslation_fr_Text767), ADR(gc_DbmTranslation_fr_Text768), ADR(gc_DbmTranslation_fr_Text769), ADR(gc_DbmTranslation_fr_Text770), ADR(gc_DbmTranslation_fr_Text771), ADR(gc_DbmTranslation_fr_Text772), ADR(gc_DbmTranslation_fr_Text773), ADR(gc_DbmTranslation_fr_Text774), ADR(gc_DbmTranslation_fr_Text775), ADR(gc_DbmTranslation_fr_Text776), ADR(gc_DbmTranslation_fr_Text777), ADR(gc_DbmTranslation_fr_Text778), ADR(gc_DbmTranslation_fr_Text779), ADR(gc_DbmTranslation_fr_Text780), ADR(gc_DbmTranslation_fr_Text781), ADR(gc_DbmTranslation_fr_Text782), ADR(gc_DbmTranslation_fr_Text783), ADR(gc_DbmTranslation_fr_Text784), ADR(gc_DbmTranslation_fr_Text785), ADR(gc_DbmTranslation_fr_Text786), ADR(gc_DbmTranslation_fr_Text787), ADR(gc_DbmTranslation_fr_Text788), ADR(gc_DbmTranslation_fr_Text789), ADR(gc_DbmTranslation_fr_Text790), ADR(gc_DbmTranslation_fr_Text791), ADR(gc_DbmTranslation_fr_Text792), ADR(gc_DbmTranslation_fr_Text793), ADR(gc_DbmTranslation_fr_Text794), ADR(gc_DbmTranslation_fr_Text795), ADR(gc_DbmTranslation_fr_Text796), ADR(gc_DbmTranslation_fr_Text797), ADR(gc_DbmTranslation_fr_Text798), ADR(gc_DbmTranslation_fr_Text799), ADR(gc_DbmTranslation_fr_Text800), ADR(gc_DbmTranslation_fr_Text801), ADR(gc_DbmTranslation_fr_Text802), ADR(gc_DbmTranslation_fr_Text803), ADR(gc_DbmTranslation_fr_Text804), ADR(gc_DbmTranslation_fr_Text805), ADR(gc_DbmTranslation_fr_Text806), ADR(gc_DbmTranslation_fr_Text807), ADR(gc_DbmTranslation_fr_Text808), ADR(gc_DbmTranslation_fr_Text809), ADR(gc_DbmTranslation_fr_Text810), ADR(gc_DbmTranslation_fr_Text811), ADR(gc_DbmTranslation_fr_Text812), ADR(gc_DbmTranslation_fr_Text813), ADR(gc_DbmTranslation_fr_Text814), ADR(gc_DbmTranslation_fr_Text815), ADR(gc_DbmTranslation_fr_Text816), ADR(gc_DbmTranslation_fr_Text817), ADR(gc_DbmTranslation_fr_Text818), ADR(gc_DbmTranslation_fr_Text819), ADR(gc_DbmTranslation_fr_Text820), ADR(gc_DbmTranslation_fr_Text821), ADR(gc_DbmTranslation_fr_Text822), ADR(gc_DbmTranslation_fr_Text823), ADR(gc_DbmTranslation_fr_Text824), ADR(gc_DbmTranslation_fr_Text825), ADR(gc_DbmTranslation_fr_Text826), ADR(gc_DbmTranslation_fr_Text827), ADR(gc_DbmTranslation_fr_Text828), ADR(gc_DbmTranslation_fr_Text829), ADR(gc_DbmTranslation_fr_Text830), ADR(gc_DbmTranslation_fr_Text831), ADR(gc_DbmTranslation_fr_Text832), ADR(gc_DbmTranslation_fr_Text833), ADR(gc_DbmTranslation_fr_Text834), ADR(gc_DbmTranslation_fr_Text835), ADR(gc_DbmTranslation_fr_Text836), ADR(gc_DbmTranslation_fr_Text837), ADR(gc_DbmTranslation_fr_Text838), ADR(gc_DbmTranslation_fr_Text839), ADR(gc_DbmTranslation_fr_Text840), ADR(gc_DbmTranslation_fr_Text841), ADR(gc_DbmTranslation_fr_Text842), ADR(gc_DbmTranslation_fr_Text843), ADR(gc_DbmTranslation_fr_Text844), ADR(gc_DbmTranslation_fr_Text845), ADR(gc_DbmTranslation_fr_Text846), ADR(gc_DbmTranslation_fr_Text847), ADR(gc_DbmTranslation_fr_Text848), ADR(gc_DbmTranslation_fr_Text849), ADR(gc_DbmTranslation_fr_Text850), ADR(gc_DbmTranslation_fr_Text851), ADR(gc_DbmTranslation_fr_Text852), ADR(gc_DbmTranslation_fr_Text853), ADR(gc_DbmTranslation_fr_Text854), ADR(gc_DbmTranslation_fr_Text855), ADR(gc_DbmTranslation_fr_Text856), ADR(gc_DbmTranslation_fr_Text857), ADR(gc_DbmTranslation_fr_Text858), ADR(gc_DbmTranslation_fr_Text859), ADR(gc_DbmTranslation_fr_Text860), ADR(gc_DbmTranslation_fr_Text861), ADR(gc_DbmTranslation_fr_Text862), ADR(gc_DbmTranslation_fr_Text863), ADR(gc_DbmTranslation_fr_Text864), ADR(gc_DbmTranslation_fr_Text865), ADR(gc_DbmTranslation_fr_Text866), ADR(gc_DbmTranslation_fr_Text867), ADR(gc_DbmTranslation_fr_Text868), ADR(gc_DbmTranslation_fr_Text869), ADR(gc_DbmTranslation_fr_Text870), ADR(gc_DbmTranslation_fr_Text871), ADR(gc_DbmTranslation_fr_Text872), ADR(gc_DbmTranslation_fr_Text873), ADR(gc_DbmTranslation_fr_Text874), ADR(gc_DbmTranslation_fr_Text875), ADR(gc_DbmTranslation_fr_Text876), ADR(gc_DbmTranslation_fr_Text877), ADR(gc_DbmTranslation_fr_Text878), ADR(gc_DbmTranslation_fr_Text879), ADR(gc_DbmTranslation_fr_Text880), ADR(gc_DbmTranslation_fr_Text881), ADR(gc_DbmTranslation_fr_Text882), ADR(gc_DbmTranslation_fr_Text883), ADR(gc_DbmTranslation_fr_Text884), ADR(gc_DbmTranslation_fr_Text885), ADR(gc_DbmTranslation_fr_Text886), ADR(gc_DbmTranslation_fr_Text887), ADR(gc_DbmTranslation_fr_Text888), ADR(gc_DbmTranslation_fr_Text889), ADR(gc_DbmTranslation_fr_Text890), ADR(gc_DbmTranslation_fr_Text891), ADR(gc_DbmTranslation_fr_Text892), ADR(gc_DbmTranslation_fr_Text893), ADR(gc_DbmTranslation_fr_Text894), ADR(gc_DbmTranslation_fr_Text895), ADR(gc_DbmTranslation_fr_Text896), ADR(gc_DbmTranslation_fr_Text897), ADR(gc_DbmTranslation_fr_Text898), ADR(gc_DbmTranslation_fr_Text899), ADR(gc_DbmTranslation_fr_Text900), ADR(gc_DbmTranslation_fr_Text901), ADR(gc_DbmTranslation_fr_Text902), ADR(gc_DbmTranslation_fr_Text903), ADR(gc_DbmTranslation_fr_Text904), ADR(gc_DbmTranslation_fr_Text905), ADR(gc_DbmTranslation_fr_Text906), ADR(gc_DbmTranslation_fr_Text907), ADR(gc_DbmTranslation_fr_Text908), ADR(gc_DbmTranslation_fr_Text909), ADR(gc_DbmTranslation_fr_Text910), ADR(gc_DbmTranslation_fr_Text911), ADR(gc_DbmTranslation_fr_Text912), ADR(gc_DbmTranslation_fr_Text913), ADR(gc_DbmTranslation_fr_Text914), ADR(gc_DbmTranslation_fr_Text915), ADR(gc_DbmTranslation_fr_Text916), ADR(gc_DbmTranslation_fr_Text917), ADR(gc_DbmTranslation_fr_Text918), ADR(gc_DbmTranslation_fr_Text919), ADR(gc_DbmTranslation_fr_Text920), ADR(gc_DbmTranslation_fr_Text921), ADR(gc_DbmTranslation_fr_Text922), ADR(gc_DbmTranslation_fr_Text923), ADR(gc_DbmTranslation_fr_Text924), ADR(gc_DbmTranslation_fr_Text925), ADR(gc_DbmTranslation_fr_Text926), ADR(gc_DbmTranslation_fr_Text927), ADR(gc_DbmTranslation_fr_Text928), ADR(gc_DbmTranslation_fr_Text929), ADR(gc_DbmTranslation_fr_Text930), ADR(gc_DbmTranslation_fr_Text931), ADR(gc_DbmTranslation_fr_Text932), ADR(gc_DbmTranslation_fr_Text933), ADR(gc_DbmTranslation_fr_Text934), ADR(gc_DbmTranslation_fr_Text935), ADR(gc_DbmTranslation_fr_Text936), ADR(gc_DbmTranslation_fr_Text937), ADR(gc_DbmTranslation_fr_Text938), ADR(gc_DbmTranslation_fr_Text939), ADR(gc_DbmTranslation_fr_Text940), ADR(gc_DbmTranslation_fr_Text941), ADR(gc_DbmTranslation_fr_Text942), ADR(gc_DbmTranslation_fr_Text943), ADR(gc_DbmTranslation_fr_Text944), ADR(gc_DbmTranslation_fr_Text945), ADR(gc_DbmTranslation_fr_Text946), ADR(gc_DbmTranslation_fr_Text947), ADR(gc_DbmTranslation_fr_Text948), ADR(gc_DbmTranslation_fr_Text949), ADR(gc_DbmTranslation_fr_Text950), ADR(gc_DbmTranslation_fr_Text951), ADR(gc_DbmTranslation_fr_Text952), ADR(gc_DbmTranslation_fr_Text953), ADR(gc_DbmTranslation_fr_Text954), ADR(gc_DbmTranslation_fr_Text955), ADR(gc_DbmTranslation_fr_Text956), ADR(gc_DbmTranslation_fr_Text957), ADR(gc_DbmTranslation_fr_Text958), ADR(gc_DbmTranslation_fr_Text959), ADR(gc_DbmTranslation_fr_Text960), ADR(gc_DbmTranslation_fr_Text961), ADR(gc_DbmTranslation_fr_Text962), ADR(gc_DbmTranslation_fr_Text963), ADR(gc_DbmTranslation_fr_Text964), ADR(gc_DbmTranslation_fr_Text965), ADR(gc_DbmTranslation_fr_Text966), ADR(gc_DbmTranslation_fr_Text967), ADR(gc_DbmTranslation_fr_Text968), ADR(gc_DbmTranslation_fr_Text969), ADR(gc_DbmTranslation_fr_Text970), ADR(gc_DbmTranslation_fr_Text971), ADR(gc_DbmTranslation_fr_Text972), ADR(gc_DbmTranslation_fr_Text973), ADR(gc_DbmTranslation_fr_Text974), ADR(gc_DbmTranslation_fr_Text975), ADR(gc_DbmTranslation_fr_Text976), ADR(gc_DbmTranslation_fr_Text977), ADR(gc_DbmTranslation_fr_Text978), ADR(gc_DbmTranslation_fr_Text979), ADR(gc_DbmTranslation_fr_Text980), ADR(gc_DbmTranslation_fr_Text981), ADR(gc_DbmTranslation_fr_Text982), ADR(gc_DbmTranslation_fr_Text983), ADR(gc_DbmTranslation_fr_Text984), ADR(gc_DbmTranslation_fr_Text985), ADR(gc_DbmTranslation_fr_Text986), ADR(gc_DbmTranslation_fr_Text987), ADR(gc_DbmTranslation_fr_Text988), ADR(gc_DbmTranslation_fr_Text989), ADR(gc_DbmTranslation_fr_Text990), ADR(gc_DbmTranslation_fr_Text991), ADR(gc_DbmTranslation_fr_Text992), ADR(gc_DbmTranslation_fr_Text993), ADR(gc_DbmTranslation_fr_Text994), ADR(gc_DbmTranslation_fr_Text995), ADR(gc_DbmTranslation_fr_Text996), ADR(gc_DbmTranslation_fr_Text997), ADR(gc_DbmTranslation_fr_Text998), ADR(gc_DbmTranslation_fr_Text999), ADR(gc_DbmTranslation_fr_Text1000), ADR(gc_DbmTranslation_fr_Text1001), ADR(gc_DbmTranslation_fr_Text1002), ADR(gc_DbmTranslation_fr_Text1003), ADR(gc_DbmTranslation_fr_Text1004), ADR(gc_DbmTranslation_fr_Text1005), ADR(gc_DbmTranslation_fr_Text1006), ADR(gc_DbmTranslation_fr_Text1007), ADR(gc_DbmTranslation_fr_Text1008), ADR(gc_DbmTranslation_fr_Text1009), ADR(gc_DbmTranslation_fr_Text1010), ADR(gc_DbmTranslation_fr_Text1011), ADR(gc_DbmTranslation_fr_Text1012), ADR(gc_DbmTranslation_fr_Text1013), ADR(gc_DbmTranslation_fr_Text1014), ADR(gc_DbmTranslation_fr_Text1015), ADR(gc_DbmTranslation_fr_Text1016), ADR(gc_DbmTranslation_fr_Text1017), ADR(gc_DbmTranslation_fr_Text1018), ADR(gc_DbmTranslation_fr_Text1019), ADR(gc_DbmTranslation_fr_Text1020), ADR(gc_DbmTranslation_fr_Text1021), ADR(gc_DbmTranslation_fr_Text1022), ADR(gc_DbmTranslation_fr_Text1023), ADR(gc_DbmTranslation_fr_Text1024), ADR(gc_DbmTranslation_fr_Text1025), ADR(gc_DbmTranslation_fr_Text1026), ADR(gc_DbmTranslation_fr_Text1027), ADR(gc_DbmTranslation_fr_Text1028), ADR(gc_DbmTranslation_fr_Text1029), ADR(gc_DbmTranslation_fr_Text1030), ADR(gc_DbmTranslation_fr_Text1031), ADR(gc_DbmTranslation_fr_Text1032), ADR(gc_DbmTranslation_fr_Text1033), ADR(gc_DbmTranslation_fr_Text1034), ADR(gc_DbmTranslation_fr_Text1035), ADR(gc_DbmTranslation_fr_Text1036), ADR(gc_DbmTranslation_fr_Text1037), ADR(gc_DbmTranslation_fr_Text1038), ADR(gc_DbmTranslation_fr_Text1039), ADR(gc_DbmTranslation_fr_Text1040), ADR(gc_DbmTranslation_fr_Text1041), ADR(gc_DbmTranslation_fr_Text1042), ADR(gc_DbmTranslation_fr_Text1043), ADR(gc_DbmTranslation_fr_Text1044), ADR(gc_DbmTranslation_fr_Text1045), ADR(gc_DbmTranslation_fr_Text1046), ADR(gc_DbmTranslation_fr_Text1047), ADR(gc_DbmTranslation_fr_Text1048), ADR(gc_DbmTranslation_fr_Text1049), ADR(gc_DbmTranslation_fr_Text1050), ADR(gc_DbmTranslation_fr_Text1051), ADR(gc_DbmTranslation_fr_Text1052), ADR(gc_DbmTranslation_fr_Text1053), ADR(gc_DbmTranslation_fr_Text1054), ADR(gc_DbmTranslation_fr_Text1055), ADR(gc_DbmTranslation_fr_Text1056), ADR(gc_DbmTranslation_fr_Text1057), ADR(gc_DbmTranslation_fr_Text1058), ADR(gc_DbmTranslation_fr_Text1059), ADR(gc_DbmTranslation_fr_Text1060), ADR(gc_DbmTranslation_fr_Text1061), ADR(gc_DbmTranslation_fr_Text1062), ADR(gc_DbmTranslation_fr_Text1063), ADR(gc_DbmTranslation_fr_Text1064), ADR(gc_DbmTranslation_fr_Text1065), ADR(gc_DbmTranslation_fr_Text1066), ADR(gc_DbmTranslation_fr_Text1067), ADR(gc_DbmTranslation_fr_Text1068), ADR(gc_DbmTranslation_fr_Text1069), ADR(gc_DbmTranslation_fr_Text1070), ADR(gc_DbmTranslation_fr_Text1071), ADR(gc_DbmTranslation_fr_Text1072), ADR(gc_DbmTranslation_fr_Text1073), ADR(gc_DbmTranslation_fr_Text1074), ADR(gc_DbmTranslation_fr_Text1075), ADR(gc_DbmTranslation_fr_Text1076), ADR(gc_DbmTranslation_fr_Text1077), ADR(gc_DbmTranslation_fr_Text1078), ADR(gc_DbmTranslation_fr_Text1079), ADR(gc_DbmTranslation_fr_Text1080), ADR(gc_DbmTranslation_fr_Text1081), ADR(gc_DbmTranslation_fr_Text1082), ADR(gc_DbmTranslation_fr_Text1083), ADR(gc_DbmTranslation_fr_Text1084), ADR(gc_DbmTranslation_fr_Text1085), ADR(gc_DbmTranslation_fr_Text1086), ADR(gc_DbmTranslation_fr_Text1087), ADR(gc_DbmTranslation_fr_Text1088), ADR(gc_DbmTranslation_fr_Text1089), ADR(gc_DbmTranslation_fr_Text1090), ADR(gc_DbmTranslation_fr_Text1091), ADR(gc_DbmTranslation_fr_Text1092), ADR(gc_DbmTranslation_fr_Text1093), ADR(gc_DbmTranslation_fr_Text1094), ADR(gc_DbmTranslation_fr_Text1095), ADR(gc_DbmTranslation_fr_Text1096), ADR(gc_DbmTranslation_fr_Text1097), ADR(gc_DbmTranslation_fr_Text1098), ADR(gc_DbmTranslation_fr_Text1099), ADR(gc_DbmTranslation_fr_Text1100), ADR(gc_DbmTranslation_fr_Text1101), ADR(gc_DbmTranslation_fr_Text1102), ADR(gc_DbmTranslation_fr_Text1103), ADR(gc_DbmTranslation_fr_Text1104), ADR(gc_DbmTranslation_fr_Text1105), ADR(gc_DbmTranslation_fr_Text1106), ADR(gc_DbmTranslation_fr_Text1107), ADR(gc_DbmTranslation_fr_Text1108), ADR(gc_DbmTranslation_fr_Text1109), ADR(gc_DbmTranslation_fr_Text1110), ADR(gc_DbmTranslation_fr_Text1111), ADR(gc_DbmTranslation_fr_Text1112), ADR(gc_DbmTranslation_fr_Text1113), ADR(gc_DbmTranslation_fr_Text1114), ADR(gc_DbmTranslation_fr_Text1115), ADR(gc_DbmTranslation_fr_Text1116), ADR(gc_DbmTranslation_fr_Text1117), ADR(gc_DbmTranslation_fr_Text1118), ADR(gc_DbmTranslation_fr_Text1119), ADR(gc_DbmTranslation_fr_Text1120), ADR(gc_DbmTranslation_fr_Text1121), ADR(gc_DbmTranslation_fr_Text1122), ADR(gc_DbmTranslation_fr_Text1123), ADR(gc_DbmTranslation_fr_Text1124), ADR(gc_DbmTranslation_fr_Text1125), ADR(gc_DbmTranslation_fr_Text1126), ADR(gc_DbmTranslation_fr_Text1127), ADR(gc_DbmTranslation_fr_Text1128), ADR(gc_DbmTranslation_fr_Text1129), ADR(gc_DbmTranslation_fr_Text1130), ADR(gc_DbmTranslation_fr_Text1131), ADR(gc_DbmTranslation_fr_Text1132), ADR(gc_DbmTranslation_fr_Text1133), ADR(gc_DbmTranslation_fr_Text1134), ADR(gc_DbmTranslation_fr_Text1135), ADR(gc_DbmTranslation_fr_Text1136), ADR(gc_DbmTranslation_fr_Text1137), ADR(gc_DbmTranslation_fr_Text1138), ADR(gc_DbmTranslation_fr_Text1139), ADR(gc_DbmTranslation_fr_Text1140), ADR(gc_DbmTranslation_fr_Text1141), ADR(gc_DbmTranslation_fr_Text1142), ADR(gc_DbmTranslation_fr_Text1143), ADR(gc_DbmTranslation_fr_Text1144), ADR(gc_DbmTranslation_fr_Text1145), ADR(gc_DbmTranslation_fr_Text1146), ADR(gc_DbmTranslation_fr_Text1147), ADR(gc_DbmTranslation_fr_Text1148), ADR(gc_DbmTranslation_fr_Text1149), ADR(gc_DbmTranslation_fr_Text1150), ADR(gc_DbmTranslation_fr_Text1151), ADR(gc_DbmTranslation_fr_Text1152), ADR(gc_DbmTranslation_fr_Text1153), ADR(gc_DbmTranslation_fr_Text1154), ADR(gc_DbmTranslation_fr_Text1155), ADR(gc_DbmTranslation_fr_Text1156), ADR(gc_DbmTranslation_fr_Text1157), ADR(gc_DbmTranslation_fr_Text1158), ADR(gc_DbmTranslation_fr_Text1159), ADR(gc_DbmTranslation_fr_Text1160), ADR(gc_DbmTranslation_fr_Text1161), ADR(gc_DbmTranslation_fr_Text1162), ADR(gc_DbmTranslation_fr_Text1163), ADR(gc_DbmTranslation_fr_Text1164), ADR(gc_DbmTranslation_fr_Text1165), ADR(gc_DbmTranslation_fr_Text1166), ADR(gc_DbmTranslation_fr_Text1167), ADR(gc_DbmTranslation_fr_Text1168), ADR(gc_DbmTranslation_fr_Text1169), ADR(gc_DbmTranslation_fr_Text1170), ADR(gc_DbmTranslation_fr_Text1171), ADR(gc_DbmTranslation_fr_Text1172), ADR(gc_DbmTranslation_fr_Text1173), ADR(gc_DbmTranslation_fr_Text1174), ADR(gc_DbmTranslation_fr_Text1175), ADR(gc_DbmTranslation_fr_Text1176), ADR(gc_DbmTranslation_fr_Text1177), ADR(gc_DbmTranslation_fr_Text1178), ADR(gc_DbmTranslation_fr_Text1179), ADR(gc_DbmTranslation_fr_Text1180), ADR(gc_DbmTranslation_fr_Text1181), ADR(gc_DbmTranslation_fr_Text1182), ADR(gc_DbmTranslation_fr_Text1183), ADR(gc_DbmTranslation_fr_Text1184), ADR(gc_DbmTranslation_fr_Text1185), ADR(gc_DbmTranslation_fr_Text1186), ADR(gc_DbmTranslation_fr_Text1187), ADR(gc_DbmTranslation_fr_Text1188), ADR(gc_DbmTranslation_fr_Text1189), ADR(gc_DbmTranslation_fr_Text1190), ADR(gc_DbmTranslation_fr_Text1191), ADR(gc_DbmTranslation_fr_Text1192), ADR(gc_DbmTranslation_fr_Text1193), ADR(gc_DbmTranslation_fr_Text1194), ADR(gc_DbmTranslation_fr_Text1195), ADR(gc_DbmTranslation_fr_Text1196), ADR(gc_DbmTranslation_fr_Text1197), ADR(gc_DbmTranslation_fr_Text1198), ADR(gc_DbmTranslation_fr_Text1199), ADR(gc_DbmTranslation_fr_Text1200), ADR(gc_DbmTranslation_fr_Text1201), ADR(gc_DbmTranslation_fr_Text1202), ADR(gc_DbmTranslation_fr_Text1203), ADR(gc_DbmTranslation_fr_Text1204), ADR(gc_DbmTranslation_fr_Text1205), ADR(gc_DbmTranslation_fr_Text1206), ADR(gc_DbmTranslation_fr_Text1207), ADR(gc_DbmTranslation_fr_Text1208), ADR(gc_DbmTranslation_fr_Text1209), ADR(gc_DbmTranslation_fr_Text1210), ADR(gc_DbmTranslation_fr_Text1211), ADR(gc_DbmTranslation_fr_Text1212), ADR(gc_DbmTranslation_fr_Text1213), ADR(gc_DbmTranslation_fr_Text1214), ADR(gc_DbmTranslation_fr_Text1215), ADR(gc_DbmTranslation_fr_Text1216), ADR(gc_DbmTranslation_fr_Text1217), ADR(gc_DbmTranslation_fr_Text1218), ADR(gc_DbmTranslation_fr_Text1219), ADR(gc_DbmTranslation_fr_Text1220), ADR(gc_DbmTranslation_fr_Text1221), ADR(gc_DbmTranslation_fr_Text1222), ADR(gc_DbmTranslation_fr_Text1223), ADR(gc_DbmTranslation_fr_Text1224), ADR(gc_DbmTranslation_fr_Text1225), ADR(gc_DbmTranslation_fr_Text1226), ADR(gc_DbmTranslation_fr_Text1227), ADR(gc_DbmTranslation_fr_Text1228), ADR(gc_DbmTranslation_fr_Text1229), ADR(gc_DbmTranslation_fr_Text1230), ADR(gc_DbmTranslation_fr_Text1231), ADR(gc_DbmTranslation_fr_Text1232), ADR(gc_DbmTranslation_fr_Text1233), ADR(gc_DbmTranslation_fr_Text1234), ADR(gc_DbmTranslation_fr_Text1235), ADR(gc_DbmTranslation_fr_Text1236), ADR(gc_DbmTranslation_fr_Text1237), ADR(gc_DbmTranslation_fr_Text1238), ADR(gc_DbmTranslation_fr_Text1239), ADR(gc_DbmTranslation_fr_Text1240), ADR(gc_DbmTranslation_fr_Text1241), ADR(gc_DbmTranslation_fr_Text1242), ADR(gc_DbmTranslation_fr_Text1243), ADR(gc_DbmTranslation_fr_Text1244), ADR(gc_DbmTranslation_fr_Text1245), ADR(gc_DbmTranslation_fr_Text1246), ADR(gc_DbmTranslation_fr_Text1247), ADR(gc_DbmTranslation_fr_Text1248), ADR(gc_DbmTranslation_fr_Text1249), ADR(gc_DbmTranslation_fr_Text1250), ADR(gc_DbmTranslation_fr_Text1251), ADR(gc_DbmTranslation_fr_Text1252), ADR(gc_DbmTranslation_fr_Text1253), ADR(gc_DbmTranslation_fr_Text1254), ADR(gc_DbmTranslation_fr_Text1255), ADR(gc_DbmTranslation_fr_Text1256), ADR(gc_DbmTranslation_fr_Text1257), ADR(gc_DbmTranslation_fr_Text1258), ADR(gc_DbmTranslation_fr_Text1259), ADR(gc_DbmTranslation_fr_Text1260), ADR(gc_DbmTranslation_fr_Text1261), ADR(gc_DbmTranslation_fr_Text1262), ADR(gc_DbmTranslation_fr_Text1263), ADR(gc_DbmTranslation_fr_Text1264), ADR(gc_DbmTranslation_fr_Text1265), ADR(gc_DbmTranslation_fr_Text1266), ADR(gc_DbmTranslation_fr_Text1267), ADR(gc_DbmTranslation_fr_Text1268), ADR(gc_DbmTranslation_fr_Text1269), ADR(gc_DbmTranslation_fr_Text1270), ADR(gc_DbmTranslation_fr_Text1271), ADR(gc_DbmTranslation_fr_Text1272), ADR(gc_DbmTranslation_fr_Text1273), ADR(gc_DbmTranslation_fr_Text1274), ADR(gc_DbmTranslation_fr_Text1275), ADR(gc_DbmTranslation_fr_Text1276), ADR(gc_DbmTranslation_fr_Text1277), ADR(gc_DbmTranslation_fr_Text1278), ADR(gc_DbmTranslation_fr_Text1279), ADR(gc_DbmTranslation_fr_Text1280), ADR(gc_DbmTranslation_fr_Text1281), ADR(gc_DbmTranslation_fr_Text1282), ADR(gc_DbmTranslation_fr_Text1283), ADR(gc_DbmTranslation_fr_Text1284), ADR(gc_DbmTranslation_fr_Text1285), ADR(gc_DbmTranslation_fr_Text1286), ADR(gc_DbmTranslation_fr_Text1287), ADR(gc_DbmTranslation_fr_Text1288), ADR(gc_DbmTranslation_fr_Text1289), ADR(gc_DbmTranslation_fr_Text1290), ADR(gc_DbmTranslation_fr_Text1291), ADR(gc_DbmTranslation_fr_Text1292), ADR(gc_DbmTranslation_fr_Text1293), ADR(gc_DbmTranslation_fr_Text1294), ADR(gc_DbmTranslation_fr_Text1295), ADR(gc_DbmTranslation_fr_Text1296), ADR(gc_DbmTranslation_fr_Text1297), ADR(gc_DbmTranslation_fr_Text1298), ADR(gc_DbmTranslation_fr_Text1299), ADR(gc_DbmTranslation_fr_Text1300), ADR(gc_DbmTranslation_fr_Text1301), ADR(gc_DbmTranslation_fr_Text1302), ADR(gc_DbmTranslation_fr_Text1303), ADR(gc_DbmTranslation_fr_Text1304), ADR(gc_DbmTranslation_fr_Text1305), ADR(gc_DbmTranslation_fr_Text1306), ADR(gc_DbmTranslation_fr_Text1307), ADR(gc_DbmTranslation_fr_Text1308), ADR(gc_DbmTranslation_fr_Text1309), ADR(gc_DbmTranslation_fr_Text1310), ADR(gc_DbmTranslation_fr_Text1311), ADR(gc_DbmTranslation_fr_Text1312), ADR(gc_DbmTranslation_fr_Text1313), ADR(gc_DbmTranslation_fr_Text1314), ADR(gc_DbmTranslation_fr_Text1315), ADR(gc_DbmTranslation_fr_Text1316), ADR(gc_DbmTranslation_fr_Text1317), ADR(gc_DbmTranslation_fr_Text1318), ADR(gc_DbmTranslation_fr_Text1319), ADR(gc_DbmTranslation_fr_Text1320), ADR(gc_DbmTranslation_fr_Text1321), ADR(gc_DbmTranslation_fr_Text1322), ADR(gc_DbmTranslation_fr_Text1323), ADR(gc_DbmTranslation_fr_Text1324), ADR(gc_DbmTranslation_fr_Text1325), ADR(gc_DbmTranslation_fr_Text1326), ADR(gc_DbmTranslation_fr_Text1327), ADR(gc_DbmTranslation_fr_Text1328), ADR(gc_DbmTranslation_fr_Text1329), ADR(gc_DbmTranslation_fr_Text1330), ADR(gc_DbmTranslation_fr_Text1331), ADR(gc_DbmTranslation_fr_Text1332), ADR(gc_DbmTranslation_fr_Text1333), ADR(gc_DbmTranslation_fr_Text1334), ADR(gc_DbmTranslation_fr_Text1335), ADR(gc_DbmTranslation_fr_Text1336), ADR(gc_DbmTranslation_fr_Text1337), ADR(gc_DbmTranslation_fr_Text1338), ADR(gc_DbmTranslation_fr_Text1339), ADR(gc_DbmTranslation_fr_Text1340), ADR(gc_DbmTranslation_fr_Text1341), ADR(gc_DbmTranslation_fr_Text1342), ADR(gc_DbmTranslation_fr_Text1343), ADR(gc_DbmTranslation_fr_Text1344), ADR(gc_DbmTranslation_fr_Text1345), ADR(gc_DbmTranslation_fr_Text1346), ADR(gc_DbmTranslation_fr_Text1347), ADR(gc_DbmTranslation_fr_Text1348), ADR(gc_DbmTranslation_fr_Text1349), ADR(gc_DbmTranslation_fr_Text1350), ADR(gc_DbmTranslation_fr_Text1351), ADR(gc_DbmTranslation_fr_Text1352), ADR(gc_DbmTranslation_fr_Text1353), ADR(gc_DbmTranslation_fr_Text1354), ADR(gc_DbmTranslation_fr_Text1355), ADR(gc_DbmTranslation_fr_Text1356), ADR(gc_DbmTranslation_fr_Text1357), ADR(gc_DbmTranslation_fr_Text1358), ADR(gc_DbmTranslation_fr_Text1359), ADR(gc_DbmTranslation_fr_Text1360), ADR(gc_DbmTranslation_fr_Text1361), ADR(gc_DbmTranslation_fr_Text1362), ADR(gc_DbmTranslation_fr_Text1363), ADR(gc_DbmTranslation_fr_Text1364), ADR(gc_DbmTranslation_fr_Text1365), ADR(gc_DbmTranslation_fr_Text1366), ADR(gc_DbmTranslation_fr_Text1367), ADR(gc_DbmTranslation_fr_Text1368), ADR(gc_DbmTranslation_fr_Text1369), ADR(gc_DbmTranslation_fr_Text1370), ADR(gc_DbmTranslation_fr_Text1371), ADR(gc_DbmTranslation_fr_Text1372), ADR(gc_DbmTranslation_fr_Text1373), ADR(gc_DbmTranslation_fr_Text1374), ADR(gc_DbmTranslation_fr_Text1375), ADR(gc_DbmTranslation_fr_Text1376), ADR(gc_DbmTranslation_fr_Text1377), ADR(gc_DbmTranslation_fr_Text1378), ADR(gc_DbmTranslation_fr_Text1379), ADR(gc_DbmTranslation_fr_Text1380), ADR(gc_DbmTranslation_fr_Text1381), ADR(gc_DbmTranslation_fr_Text1382), ADR(gc_DbmTranslation_fr_Text1383), ADR(gc_DbmTranslation_fr_Text1384), ADR(gc_DbmTranslation_fr_Text1385), ADR(gc_DbmTranslation_fr_Text1386), ADR(gc_DbmTranslation_fr_Text1387), ADR(gc_DbmTranslation_fr_Text1388), ADR(gc_DbmTranslation_fr_Text1389), ADR(gc_DbmTranslation_fr_Text1390), ADR(gc_DbmTranslation_fr_Text1391), ADR(gc_DbmTranslation_fr_Text1392), ADR(gc_DbmTranslation_fr_Text1393), ADR(gc_DbmTranslation_fr_Text1394), ADR(gc_DbmTranslation_fr_Text1395), ADR(gc_DbmTranslation_fr_Text1396), ADR(gc_DbmTranslation_fr_Text1397), ADR(gc_DbmTranslation_fr_Text1398), ADR(gc_DbmTranslation_fr_Text1399), ADR(gc_DbmTranslation_fr_Text1400), ADR(gc_DbmTranslation_fr_Text1401), ADR(gc_DbmTranslation_fr_Text1402), ADR(gc_DbmTranslation_fr_Text1403), ADR(gc_DbmTranslation_fr_Text1404), ADR(gc_DbmTranslation_fr_Text1405), ADR(gc_DbmTranslation_fr_Text1406), ADR(gc_DbmTranslation_fr_Text1407), ADR(gc_DbmTranslation_fr_Text1408), ADR(gc_DbmTranslation_fr_Text1409), ADR(gc_DbmTranslation_fr_Text1410), ADR(gc_DbmTranslation_fr_Text1411), ADR(gc_DbmTranslation_fr_Text1412), ADR(gc_DbmTranslation_fr_Text1413), ADR(gc_DbmTranslation_fr_Text1414), ADR(gc_DbmTranslation_fr_Text1415), ADR(gc_DbmTranslation_fr_Text1416), ADR(gc_DbmTranslation_fr_Text1417), ADR(gc_DbmTranslation_fr_Text1418), ADR(gc_DbmTranslation_fr_Text1419), ADR(gc_DbmTranslation_fr_Text1420), ADR(gc_DbmTranslation_fr_Text1421), ADR(gc_DbmTranslation_fr_Text1422), ADR(gc_DbmTranslation_fr_Text1423), ADR(gc_DbmTranslation_fr_Text1424), ADR(gc_DbmTranslation_fr_Text1425), ADR(gc_DbmTranslation_fr_Text1426), ADR(gc_DbmTranslation_fr_Text1427), ADR(gc_DbmTranslation_fr_Text1428), ADR(gc_DbmTranslation_fr_Text1429), ADR(gc_DbmTranslation_fr_Text1430), ADR(gc_DbmTranslation_fr_Text1431), ADR(gc_DbmTranslation_fr_Text1432), ADR(gc_DbmTranslation_fr_Text1433), ADR(gc_DbmTranslation_fr_Text1434), ADR(gc_DbmTranslation_fr_Text1435), ADR(gc_DbmTranslation_fr_Text1436), ADR(gc_DbmTranslation_fr_Text1437), ADR(gc_DbmTranslation_fr_Text1438), ADR(gc_DbmTranslation_fr_Text1439), ADR(gc_DbmTranslation_fr_Text1440), ADR(gc_DbmTranslation_fr_Text1441), ADR(gc_DbmTranslation_fr_Text1442), ADR(gc_DbmTranslation_fr_Text1443), ADR(gc_DbmTranslation_fr_Text1444), ADR(gc_DbmTranslation_fr_Text1445), ADR(gc_DbmTranslation_fr_Text1446), ADR(gc_DbmTranslation_fr_Text1447), ADR(gc_DbmTranslation_fr_Text1448), ADR(gc_DbmTranslation_fr_Text1449), ADR(gc_DbmTranslation_fr_Text1450), ADR(gc_DbmTranslation_fr_Text1451), ADR(gc_DbmTranslation_fr_Text1452), ADR(gc_DbmTranslation_fr_Text1453), ADR(gc_DbmTranslation_fr_Text1454), ADR(gc_DbmTranslation_fr_Text1455), ADR(gc_DbmTranslation_fr_Text1456), ADR(gc_DbmTranslation_fr_Text1457), ADR(gc_DbmTranslation_fr_Text1458), ADR(gc_DbmTranslation_fr_Text1459), ADR(gc_DbmTranslation_fr_Text1460), ADR(gc_DbmTranslation_fr_Text1461), ADR(gc_DbmTranslation_fr_Text1462), ADR(gc_DbmTranslation_fr_Text1463), ADR(gc_DbmTranslation_fr_Text1464), ADR(gc_DbmTranslation_fr_Text1465), ADR(gc_DbmTranslation_fr_Text1466), ADR(gc_DbmTranslation_fr_Text1467), ADR(gc_DbmTranslation_fr_Text1468), ADR(gc_DbmTranslation_fr_Text1469), ADR(gc_DbmTranslation_fr_Text1470), ADR(gc_DbmTranslation_fr_Text1471), ADR(gc_DbmTranslation_fr_Text1472), ADR(gc_DbmTranslation_fr_Text1473), ADR(gc_DbmTranslation_fr_Text1474), ADR(gc_DbmTranslation_fr_Text1475), ADR(gc_DbmTranslation_fr_Text1476), ADR(gc_DbmTranslation_fr_Text1477), ADR(gc_DbmTranslation_fr_Text1478), ADR(gc_DbmTranslation_fr_Text1479), ADR(gc_DbmTranslation_fr_Text1480), ADR(gc_DbmTranslation_fr_Text1481), ADR(gc_DbmTranslation_fr_Text1482), ADR(gc_DbmTranslation_fr_Text1483), ADR(gc_DbmTranslation_fr_Text1484), ADR(gc_DbmTranslation_fr_Text1485), ADR(gc_DbmTranslation_fr_Text1486), ADR(gc_DbmTranslation_fr_Text1487), ADR(gc_DbmTranslation_fr_Text1488), ADR(gc_DbmTranslation_fr_Text1489), ADR(gc_DbmTranslation_fr_Text1490), ADR(gc_DbmTranslation_fr_Text1491), ADR(gc_DbmTranslation_fr_Text1492), ADR(gc_DbmTranslation_fr_Text1493), ADR(gc_DbmTranslation_fr_Text1494), ADR(gc_DbmTranslation_fr_Text1495), ADR(gc_DbmTranslation_fr_Text1496), ADR(gc_DbmTranslation_fr_Text1497), ADR(gc_DbmTranslation_fr_Text1498), ADR(gc_DbmTranslation_fr_Text1499), ADR(gc_DbmTranslation_fr_Text1500), ADR(gc_DbmTranslation_fr_Text1501), ADR(gc_DbmTranslation_fr_Text1502), ADR(gc_DbmTranslation_fr_Text1503), ADR(gc_DbmTranslation_fr_Text1504), ADR(gc_DbmTranslation_fr_Text1505), ADR(gc_DbmTranslation_fr_Text1506), ADR(gc_DbmTranslation_fr_Text1507), ADR(gc_DbmTranslation_fr_Text1508), ADR(gc_DbmTranslation_fr_Text1509), ADR(gc_DbmTranslation_fr_Text1510), ADR(gc_DbmTranslation_fr_Text1511), ADR(gc_DbmTranslation_fr_Text1512), ADR(gc_DbmTranslation_fr_Text1513), ADR(gc_DbmTranslation_fr_Text1514), ADR(gc_DbmTranslation_fr_Text1515), ADR(gc_DbmTranslation_fr_Text1516), ADR(gc_DbmTranslation_fr_Text1517), ADR(gc_DbmTranslation_fr_Text1518), ADR(gc_DbmTranslation_fr_Text1519), ADR(gc_DbmTranslation_fr_Text1520), ADR(gc_DbmTranslation_fr_Text1521), ADR(gc_DbmTranslation_fr_Text1522), ADR(gc_DbmTranslation_fr_Text1523), ADR(gc_DbmTranslation_fr_Text1524), ADR(gc_DbmTranslation_fr_Text1525), ADR(gc_DbmTranslation_fr_Text1526), ADR(gc_DbmTranslation_fr_Text1527), ADR(gc_DbmTranslation_fr_Text1528), ADR(gc_DbmTranslation_fr_Text1529), ADR(gc_DbmTranslation_fr_Text1530), ADR(gc_DbmTranslation_fr_Text1531), ADR(gc_DbmTranslation_fr_Text1532), ADR(gc_DbmTranslation_fr_Text1533), ADR(gc_DbmTranslation_fr_Text1534), ADR(gc_DbmTranslation_fr_Text1535), ADR(gc_DbmTranslation_fr_Text1536), ADR(gc_DbmTranslation_fr_Text1537), ADR(gc_DbmTranslation_fr_Text1538), ADR(gc_DbmTranslation_fr_Text1539), ADR(gc_DbmTranslation_fr_Text1540), ADR(gc_DbmTranslation_fr_Text1541), ADR(gc_DbmTranslation_fr_Text1542), ADR(gc_DbmTranslation_fr_Text1543), ADR(gc_DbmTranslation_fr_Text1544), ADR(gc_DbmTranslation_fr_Text1545), ADR(gc_DbmTranslation_fr_Text1546), ADR(gc_DbmTranslation_fr_Text1547), ADR(gc_DbmTranslation_fr_Text1548), ADR(gc_DbmTranslation_fr_Text1549), ADR(gc_DbmTranslation_fr_Text1550), ADR(gc_DbmTranslation_fr_Text1551), ADR(gc_DbmTranslation_fr_Text1552), ADR(gc_DbmTranslation_fr_Text1553), ADR(gc_DbmTranslation_fr_Text1554), ADR(gc_DbmTranslation_fr_Text1555), ADR(gc_DbmTranslation_fr_Text1556), ADR(gc_DbmTranslation_fr_Text1557), ADR(gc_DbmTranslation_fr_Text1558), ADR(gc_DbmTranslation_fr_Text1559), ADR(gc_DbmTranslation_fr_Text1560), ADR(gc_DbmTranslation_fr_Text1561), ADR(gc_DbmTranslation_fr_Text1562), ADR(gc_DbmTranslation_fr_Text1563), ADR(gc_DbmTranslation_fr_Text1564), ADR(gc_DbmTranslation_fr_Text1565), ADR(gc_DbmTranslation_fr_Text1566), ADR(gc_DbmTranslation_fr_Text1567), ADR(gc_DbmTranslation_fr_Text1568), ADR(gc_DbmTranslation_fr_Text1569), ADR(gc_DbmTranslation_fr_Text1570), ADR(gc_DbmTranslation_fr_Text1571), ADR(gc_DbmTranslation_fr_Text1572), ADR(gc_DbmTranslation_fr_Text1573), ADR(gc_DbmTranslation_fr_Text1574), ADR(gc_DbmTranslation_fr_Text1575), ADR(gc_DbmTranslation_fr_Text1576), ADR(gc_DbmTranslation_fr_Text1577), ADR(gc_DbmTranslation_fr_Text1578), ADR(gc_DbmTranslation_fr_Text1579), ADR(gc_DbmTranslation_fr_Text1580), ADR(gc_DbmTranslation_fr_Text1581), ADR(gc_DbmTranslation_fr_Text1582), ADR(gc_DbmTranslation_fr_Text1583), ADR(gc_DbmTranslation_fr_Text1584), ADR(gc_DbmTranslation_fr_Text1585), ADR(gc_DbmTranslation_fr_Text1586), ADR(gc_DbmTranslation_fr_Text1587), ADR(gc_DbmTranslation_fr_Text1588), ADR(gc_DbmTranslation_fr_Text1589), ADR(gc_DbmTranslation_fr_Text1590), ADR(gc_DbmTranslation_fr_Text1591), ADR(gc_DbmTranslation_fr_Text1592), ADR(gc_DbmTranslation_fr_Text1593), ADR(gc_DbmTranslation_fr_Text1594), ADR(gc_DbmTranslation_fr_Text1595), ADR(gc_DbmTranslation_fr_Text1596), ADR(gc_DbmTranslation_fr_Text1597), ADR(gc_DbmTranslation_fr_Text1598), ADR(gc_DbmTranslation_fr_Text1599), ADR(gc_DbmTranslation_fr_Text1600), ADR(gc_DbmTranslation_fr_Text1601), ADR(gc_DbmTranslation_fr_Text1602), ADR(gc_DbmTranslation_fr_Text1603), ADR(gc_DbmTranslation_fr_Text1604), ADR(gc_DbmTranslation_fr_Text1605), ADR(gc_DbmTranslation_fr_Text1606), ADR(gc_DbmTranslation_fr_Text1607), ADR(gc_DbmTranslation_fr_Text1608), ADR(gc_DbmTranslation_fr_Text1609), ADR(gc_DbmTranslation_fr_Text1610), ADR(gc_DbmTranslation_fr_Text1611), ADR(gc_DbmTranslation_fr_Text1612), ADR(gc_DbmTranslation_fr_Text1613), ADR(gc_DbmTranslation_fr_Text1614), ADR(gc_DbmTranslation_fr_Text1615), ADR(gc_DbmTranslation_fr_Text1616), ADR(gc_DbmTranslation_fr_Text1617), ADR(gc_DbmTranslation_fr_Text1618), ADR(gc_DbmTranslation_fr_Text1619), ADR(gc_DbmTranslation_fr_Text1620), ADR(gc_DbmTranslation_fr_Text1621), ADR(gc_DbmTranslation_fr_Text1622), ADR(gc_DbmTranslation_fr_Text1623), ADR(gc_DbmTranslation_fr_Text1624), ADR(gc_DbmTranslation_fr_Text1625), ADR(gc_DbmTranslation_fr_Text1626), ADR(gc_DbmTranslation_fr_Text1627), ADR(gc_DbmTranslation_fr_Text1628), ADR(gc_DbmTranslation_fr_Text1629), ADR(gc_DbmTranslation_fr_Text1630), ADR(gc_DbmTranslation_fr_Text1631), ADR(gc_DbmTranslation_fr_Text1632), ADR(gc_DbmTranslation_fr_Text1633), ADR(gc_DbmTranslation_fr_Text1634), ADR(gc_DbmTranslation_fr_Text1635), ADR(gc_DbmTranslation_fr_Text1636), ADR(gc_DbmTranslation_fr_Text1637), ADR(gc_DbmTranslation_fr_Text1638), ADR(gc_DbmTranslation_fr_Text1639), ADR(gc_DbmTranslation_fr_Text1640), ADR(gc_DbmTranslation_fr_Text1641), ADR(gc_DbmTranslation_fr_Text1642), ADR(gc_DbmTranslation_fr_Text1643), ADR(gc_DbmTranslation_fr_Text1644), ADR(gc_DbmTranslation_fr_Text1645), ADR(gc_DbmTranslation_fr_Text1646), ADR(gc_DbmTranslation_fr_Text1647), ADR(gc_DbmTranslation_fr_Text1648), ADR(gc_DbmTranslation_fr_Text1649), ADR(gc_DbmTranslation_fr_Text1650), ADR(gc_DbmTranslation_fr_Text1651), ADR(gc_DbmTranslation_fr_Text1652), ADR(gc_DbmTranslation_fr_Text1653), ADR(gc_DbmTranslation_fr_Text1654), ADR(gc_DbmTranslation_fr_Text1655), ADR(gc_DbmTranslation_fr_Text1656), ADR(gc_DbmTranslation_fr_Text1657), ADR(gc_DbmTranslation_fr_Text1658), ADR(gc_DbmTranslation_fr_Text1659), ADR(gc_DbmTranslation_fr_Text1660), ADR(gc_DbmTranslation_fr_Text1661), ADR(gc_DbmTranslation_fr_Text1662), ADR(gc_DbmTranslation_fr_Text1663), ADR(gc_DbmTranslation_fr_Text1664), ADR(gc_DbmTranslation_fr_Text1665), ADR(gc_DbmTranslation_fr_Text1666), ADR(gc_DbmTranslation_fr_Text1667), ADR(gc_DbmTranslation_fr_Text1668), ADR(gc_DbmTranslation_fr_Text1669), ADR(gc_DbmTranslation_fr_Text1670), ADR(gc_DbmTranslation_fr_Text1671), ADR(gc_DbmTranslation_fr_Text1672), ADR(gc_DbmTranslation_fr_Text1673), ADR(gc_DbmTranslation_fr_Text1674), ADR(gc_DbmTranslation_fr_Text1675), ADR(gc_DbmTranslation_fr_Text1676), ADR(gc_DbmTranslation_fr_Text1677), ADR(gc_DbmTranslation_fr_Text1678), ADR(gc_DbmTranslation_fr_Text1679), ADR(gc_DbmTranslation_fr_Text1680), ADR(gc_DbmTranslation_fr_Text1681), ADR(gc_DbmTranslation_fr_Text1682), ADR(gc_DbmTranslation_fr_Text1683), ADR(gc_DbmTranslation_fr_Text1684), ADR(gc_DbmTranslation_fr_Text1685), ADR(gc_DbmTranslation_fr_Text1686), ADR(gc_DbmTranslation_fr_Text1687), ADR(gc_DbmTranslation_fr_Text1688), ADR(gc_DbmTranslation_fr_Text1689), ADR(gc_DbmTranslation_fr_Text1690), ADR(gc_DbmTranslation_fr_Text1691), ADR(gc_DbmTranslation_fr_Text1692), ADR(gc_DbmTranslation_fr_Text1693), ADR(gc_DbmTranslation_fr_Text1694), ADR(gc_DbmTranslation_fr_Text1695), ADR(gc_DbmTranslation_fr_Text1696), ADR(gc_DbmTranslation_fr_Text1697), ADR(gc_DbmTranslation_fr_Text1698), ADR(gc_DbmTranslation_fr_Text1699), ADR(gc_DbmTranslation_fr_Text1700), ADR(gc_DbmTranslation_fr_Text1701), ADR(gc_DbmTranslation_fr_Text1702), ADR(gc_DbmTranslation_fr_Text1703), ADR(gc_DbmTranslation_fr_Text1704), ADR(gc_DbmTranslation_fr_Text1705), ADR(gc_DbmTranslation_fr_Text1706), ADR(gc_DbmTranslation_fr_Text1707), ADR(gc_DbmTranslation_fr_Text1708), ADR(gc_DbmTranslation_fr_Text1709), ADR(gc_DbmTranslation_fr_Text1710), ADR(gc_DbmTranslation_fr_Text1711), ADR(gc_DbmTranslation_fr_Text1712), ADR(gc_DbmTranslation_fr_Text1713), ADR(gc_DbmTranslation_fr_Text1714), ADR(gc_DbmTranslation_fr_Text1715), ADR(gc_DbmTranslation_fr_Text1716), ADR(gc_DbmTranslation_fr_Text1717), ADR(gc_DbmTranslation_fr_Text1718), ADR(gc_DbmTranslation_fr_Text1719), ADR(gc_DbmTranslation_fr_Text1720), ADR(gc_DbmTranslation_fr_Text1721), ADR(gc_DbmTranslation_fr_Text1722), ADR(gc_DbmTranslation_fr_Text1723), ADR(gc_DbmTranslation_fr_Text1724), ADR(gc_DbmTranslation_fr_Text1725), ADR(gc_DbmTranslation_fr_Text1726), ADR(gc_DbmTranslation_fr_Text1727), ADR(gc_DbmTranslation_fr_Text1728), ADR(gc_DbmTranslation_fr_Text1729), ADR(gc_DbmTranslation_fr_Text1730), ADR(gc_DbmTranslation_fr_Text1731), ADR(gc_DbmTranslation_fr_Text1732), ADR(gc_DbmTranslation_fr_Text1733), ADR(gc_DbmTranslation_fr_Text1734), ADR(gc_DbmTranslation_fr_Text1735), ADR(gc_DbmTranslation_fr_Text1736), ADR(gc_DbmTranslation_fr_Text1737), ADR(gc_DbmTranslation_fr_Text1738), ADR(gc_DbmTranslation_fr_Text1739), ADR(gc_DbmTranslation_fr_Text1740), ADR(gc_DbmTranslation_fr_Text1741), ADR(gc_DbmTranslation_fr_Text1742), ADR(gc_DbmTranslation_fr_Text1743), ADR(gc_DbmTranslation_fr_Text1744), ADR(gc_DbmTranslation_fr_Text1745), ADR(gc_DbmTranslation_fr_Text1746), ADR(gc_DbmTranslation_fr_Text1747), ADR(gc_DbmTranslation_fr_Text1748), ADR(gc_DbmTranslation_fr_Text1749), ADR(gc_DbmTranslation_fr_Text1750), ADR(gc_DbmTranslation_fr_Text1751), ADR(gc_DbmTranslation_fr_Text1752), ADR(gc_DbmTranslation_fr_Text1753), ADR(gc_DbmTranslation_fr_Text1754), ADR(gc_DbmTranslation_fr_Text1755), ADR(gc_DbmTranslation_fr_Text1756), ADR(gc_DbmTranslation_fr_Text1757), ADR(gc_DbmTranslation_fr_Text1758), ADR(gc_DbmTranslation_fr_Text1759), ADR(gc_DbmTranslation_fr_Text1760), ADR(gc_DbmTranslation_fr_Text1761), ADR(gc_DbmTranslation_fr_Text1762), ADR(gc_DbmTranslation_fr_Text1763), ADR(gc_DbmTranslation_fr_Text1764), ADR(gc_DbmTranslation_fr_Text1765), ADR(gc_DbmTranslation_fr_Text1766), ADR(gc_DbmTranslation_fr_Text1767), ADR(gc_DbmTranslation_fr_Text1768), ADR(gc_DbmTranslation_fr_Text1769), ADR(gc_DbmTranslation_fr_Text1770), ADR(gc_DbmTranslation_fr_Text1771), ADR(gc_DbmTranslation_fr_Text1772), ADR(gc_DbmTranslation_fr_Text1773), ADR(gc_DbmTranslation_fr_Text1774), ADR(gc_DbmTranslation_fr_Text1775), ADR(gc_DbmTranslation_fr_Text1776), ADR(gc_DbmTranslation_fr_Text1777), ADR(gc_DbmTranslation_fr_Text1778), ADR(gc_DbmTranslation_fr_Text1779), ADR(gc_DbmTranslation_fr_Text1780), ADR(gc_DbmTranslation_fr_Text1781), ADR(gc_DbmTranslation_fr_Text1782), ADR(gc_DbmTranslation_fr_Text1783), ADR(gc_DbmTranslation_fr_Text1784), ADR(gc_DbmTranslation_fr_Text1785), ADR(gc_DbmTranslation_fr_Text1786), ADR(gc_DbmTranslation_fr_Text1787), ADR(gc_DbmTranslation_fr_Text1788), ADR(gc_DbmTranslation_fr_Text1789), ADR(gc_DbmTranslation_fr_Text1790), ADR(gc_DbmTranslation_fr_Text1791), ADR(gc_DbmTranslation_fr_Text1792), ADR(gc_DbmTranslation_fr_Text1793), ADR(gc_DbmTranslation_fr_Text1794), ADR(gc_DbmTranslation_fr_Text1795), ADR(gc_DbmTranslation_fr_Text1796), ADR(gc_DbmTranslation_fr_Text1797), ADR(gc_DbmTranslation_fr_Text1798), ADR(gc_DbmTranslation_fr_Text1799), ADR(gc_DbmTranslation_fr_Text1800), ADR(gc_DbmTranslation_fr_Text1801), ADR(gc_DbmTranslation_fr_Text1802), ADR(gc_DbmTranslation_fr_Text1803), ADR(gc_DbmTranslation_fr_Text1804), ADR(gc_DbmTranslation_fr_Text1805), ADR(gc_DbmTranslation_fr_Text1806), ADR(gc_DbmTranslation_fr_Text1807), ADR(gc_DbmTranslation_fr_Text1808), ADR(gc_DbmTranslation_fr_Text1809), ADR(gc_DbmTranslation_fr_Text1810), ADR(gc_DbmTranslation_fr_Text1811), ADR(gc_DbmTranslation_fr_Text1812), ADR(gc_DbmTranslation_fr_Text1813), ADR(gc_DbmTranslation_fr_Text1814), ADR(gc_DbmTranslation_fr_Text1815), ADR(gc_DbmTranslation_fr_Text1816), ADR(gc_DbmTranslation_fr_Text1817), ADR(gc_DbmTranslation_fr_Text1818), ADR(gc_DbmTranslation_fr_Text1819), ADR(gc_DbmTranslation_fr_Text1820), ADR(gc_DbmTranslation_fr_Text1821), ADR(gc_DbmTranslation_fr_Text1822), ADR(gc_DbmTranslation_fr_Text1823), ADR(gc_DbmTranslation_fr_Text1824), ADR(gc_DbmTranslation_fr_Text1825), ADR(gc_DbmTranslation_fr_Text1826), ADR(gc_DbmTranslation_fr_Text1827), ADR(gc_DbmTranslation_fr_Text1828), ADR(gc_DbmTranslation_fr_Text1829), ADR(gc_DbmTranslation_fr_Text1830), ADR(gc_DbmTranslation_fr_Text1831), ADR(gc_DbmTranslation_fr_Text1832), ADR(gc_DbmTranslation_fr_Text1833), ADR(gc_DbmTranslation_fr_Text1834), ADR(gc_DbmTranslation_fr_Text1835), ADR(gc_DbmTranslation_fr_Text1836), ADR(gc_DbmTranslation_fr_Text1837), ADR(gc_DbmTranslation_fr_Text1838), ADR(gc_DbmTranslation_fr_Text1839), ADR(gc_DbmTranslation_fr_Text1840), ADR(gc_DbmTranslation_fr_Text1841), ADR(gc_DbmTranslation_fr_Text1842), ADR(gc_DbmTranslation_fr_Text1843), ADR(gc_DbmTranslation_fr_Text1844), ADR(gc_DbmTranslation_fr_Text1845), ADR(gc_DbmTranslation_fr_Text1846), ADR(gc_DbmTranslation_fr_Text1847), ADR(gc_DbmTranslation_fr_Text1848), ADR(gc_DbmTranslation_fr_Text1849), ADR(gc_DbmTranslation_fr_Text1850), ADR(gc_DbmTranslation_fr_Text1851), ADR(gc_DbmTranslation_fr_Text1852), ADR(gc_DbmTranslation_fr_Text1853), ADR(gc_DbmTranslation_fr_Text1854), ADR(gc_DbmTranslation_fr_Text1855), ADR(gc_DbmTranslation_fr_Text1856), ADR(gc_DbmTranslation_fr_Text1857), ADR(gc_DbmTranslation_fr_Text1858), ADR(gc_DbmTranslation_fr_Text1859), ADR(gc_DbmTranslation_fr_Text1860), ADR(gc_DbmTranslation_fr_Text1861), ADR(gc_DbmTranslation_fr_Text1862), ADR(gc_DbmTranslation_fr_Text1863), ADR(gc_DbmTranslation_fr_Text1864), ADR(gc_DbmTranslation_fr_Text1865), ADR(gc_DbmTranslation_fr_Text1866), ADR(gc_DbmTranslation_fr_Text1867), ADR(gc_DbmTranslation_fr_Text1868), ADR(gc_DbmTranslation_fr_Text1869), ADR(gc_DbmTranslation_fr_Text1870), ADR(gc_DbmTranslation_fr_Text1871), ADR(gc_DbmTranslation_fr_Text1872), ADR(gc_DbmTranslation_fr_Text1873), ADR(gc_DbmTranslation_fr_Text1874), ADR(gc_DbmTranslation_fr_Text1875), ADR(gc_DbmTranslation_fr_Text1876), ADR(gc_DbmTranslation_fr_Text1877), ADR(gc_DbmTranslation_fr_Text1878), ADR(gc_DbmTranslation_fr_Text1879), ADR(gc_DbmTranslation_fr_Text1880), ADR(gc_DbmTranslation_fr_Text1881), ADR(gc_DbmTranslation_fr_Text1882), ADR(gc_DbmTranslation_fr_Text1883), ADR(gc_DbmTranslation_fr_Text1884), ADR(gc_DbmTranslation_fr_Text1885), ADR(gc_DbmTranslation_fr_Text1886), ADR(gc_DbmTranslation_fr_Text1887), ADR(gc_DbmTranslation_fr_Text1888), ADR(gc_DbmTranslation_fr_Text1889), ADR(gc_DbmTranslation_fr_Text1890), ADR(gc_DbmTranslation_fr_Text1891), ADR(gc_DbmTranslation_fr_Text1892), ADR(gc_DbmTranslation_fr_Text1893), ADR(gc_DbmTranslation_fr_Text1894), ADR(gc_DbmTranslation_fr_Text1895), ADR(gc_DbmTranslation_fr_Text1896), ADR(gc_DbmTranslation_fr_Text1897), ADR(gc_DbmTranslation_fr_Text1898), ADR(gc_DbmTranslation_fr_Text1899), ADR(gc_DbmTranslation_fr_Text1900), ADR(gc_DbmTranslation_fr_Text1901), ADR(gc_DbmTranslation_fr_Text1902), ADR(gc_DbmTranslation_fr_Text1903), ADR(gc_DbmTranslation_fr_Text1904), ADR(gc_DbmTranslation_fr_Text1905), ADR(gc_DbmTranslation_fr_Text1906), ADR(gc_DbmTranslation_fr_Text1907), ADR(gc_DbmTranslation_fr_Text1908), ADR(gc_DbmTranslation_fr_Text1909), ADR(gc_DbmTranslation_fr_Text1910), ADR(gc_DbmTranslation_fr_Text1911), ADR(gc_DbmTranslation_fr_Text1912), ADR(gc_DbmTranslation_fr_Text1913), ADR(gc_DbmTranslation_fr_Text1914), ADR(gc_DbmTranslation_fr_Text1915), ADR(gc_DbmTranslation_fr_Text1916), ADR(gc_DbmTranslation_fr_Text1917), ADR(gc_DbmTranslation_fr_Text1918), ADR(gc_DbmTranslation_fr_Text1919), ADR(gc_DbmTranslation_fr_Text1920), ADR(gc_DbmTranslation_fr_Text1921), ADR(gc_DbmTranslation_fr_Text1922), ADR(gc_DbmTranslation_fr_Text1923), ADR(gc_DbmTranslation_fr_Text1924), ADR(gc_DbmTranslation_fr_Text1925), ADR(gc_DbmTranslation_fr_Text1926), ADR(gc_DbmTranslation_fr_Text1927), ADR(gc_DbmTranslation_fr_Text1928), ADR(gc_DbmTranslation_fr_Text1929), ADR(gc_DbmTranslation_fr_Text1930), ADR(gc_DbmTranslation_fr_Text1931), ADR(gc_DbmTranslation_fr_Text1932), ADR(gc_DbmTranslation_fr_Text1933), ADR(gc_DbmTranslation_fr_Text1934), ADR(gc_DbmTranslation_fr_Text1935), ADR(gc_DbmTranslation_fr_Text1936), ADR(gc_DbmTranslation_fr_Text1937), ADR(gc_DbmTranslation_fr_Text1938), ADR(gc_DbmTranslation_fr_Text1939), ADR(gc_DbmTranslation_fr_Text1940), ADR(gc_DbmTranslation_fr_Text1941), ADR(gc_DbmTranslation_fr_Text1942), ADR(gc_DbmTranslation_fr_Text1943), ADR(gc_DbmTranslation_fr_Text1944), ADR(gc_DbmTranslation_fr_Text1945), ADR(gc_DbmTranslation_fr_Text1946), ADR(gc_DbmTranslation_fr_Text1947), ADR(gc_DbmTranslation_fr_Text1948), ADR(gc_DbmTranslation_fr_Text1949), ADR(gc_DbmTranslation_fr_Text1950), ADR(gc_DbmTranslation_fr_Text1951), ADR(gc_DbmTranslation_fr_Text1952), ADR(gc_DbmTranslation_fr_Text1953), ADR(gc_DbmTranslation_fr_Text1954), ADR(gc_DbmTranslation_fr_Text1955), ADR(gc_DbmTranslation_fr_Text1956), ADR(gc_DbmTranslation_fr_Text1957), ADR(gc_DbmTranslation_fr_Text1958), ADR(gc_DbmTranslation_fr_Text1959), ADR(gc_DbmTranslation_fr_Text1960), ADR(gc_DbmTranslation_fr_Text1961), ADR(gc_DbmTranslation_fr_Text1962), ADR(gc_DbmTranslation_fr_Text1963), ADR(gc_DbmTranslation_fr_Text1964), ADR(gc_DbmTranslation_fr_Text1965), ADR(gc_DbmTranslation_fr_Text1966), ADR(gc_DbmTranslation_fr_Text1967), ADR(gc_DbmTranslation_fr_Text1968), ADR(gc_DbmTranslation_fr_Text1969), ADR(gc_DbmTranslation_fr_Text1970), ADR(gc_DbmTranslation_fr_Text1971), ADR(gc_DbmTranslation_fr_Text1972), ADR(gc_DbmTranslation_fr_Text1973), ADR(gc_DbmTranslation_fr_Text1974), ADR(gc_DbmTranslation_fr_Text1975), ADR(gc_DbmTranslation_fr_Text1976), ADR(gc_DbmTranslation_fr_Text1977), ADR(gc_DbmTranslation_fr_Text1978), ADR(gc_DbmTranslation_fr_Text1979), ADR(gc_DbmTranslation_fr_Text1980), ADR(gc_DbmTranslation_fr_Text1981), ADR(gc_DbmTranslation_fr_Text1982), ADR(gc_DbmTranslation_fr_Text1983), ADR(gc_DbmTranslation_fr_Text1984), ADR(gc_DbmTranslation_fr_Text1985), ADR(gc_DbmTranslation_fr_Text1986), ADR(gc_DbmTranslation_fr_Text1987), ADR(gc_DbmTranslation_fr_Text1988), ADR(gc_DbmTranslation_fr_Text1989), ADR(gc_DbmTranslation_fr_Text1990), ADR(gc_DbmTranslation_fr_Text1991), ADR(gc_DbmTranslation_fr_Text1992), ADR(gc_DbmTranslation_fr_Text1993), ADR(gc_DbmTranslation_fr_Text1994), ADR(gc_DbmTranslation_fr_Text1995), ADR(gc_DbmTranslation_fr_Text1996), ADR(gc_DbmTranslation_fr_Text1997), ADR(gc_DbmTranslation_fr_Text1998), ADR(gc_DbmTranslation_fr_Text1999), ADR(gc_DbmTranslation_fr_Text2000), ADR(gc_DbmTranslation_fr_Text2001), ADR(gc_DbmTranslation_fr_Text2002), ADR(gc_DbmTranslation_fr_Text2003), ADR(gc_DbmTranslation_fr_Text2004), ADR(gc_DbmTranslation_fr_Text2005), ADR(gc_DbmTranslation_fr_Text2006), ADR(gc_DbmTranslation_fr_Text2007), ADR(gc_DbmTranslation_fr_Text2008), ADR(gc_DbmTranslation_fr_Text2009), ADR(gc_DbmTranslation_fr_Text2010), ADR(gc_DbmTranslation_fr_Text2011), ADR(gc_DbmTranslation_fr_Text2012), ADR(gc_DbmTranslation_fr_Text2013), ADR(gc_DbmTranslation_fr_Text2014), ADR(gc_DbmTranslation_fr_Text2015), ADR(gc_DbmTranslation_fr_Text2016), ADR(gc_DbmTranslation_fr_Text2017), ADR(gc_DbmTranslation_fr_Text2018), ADR(gc_DbmTranslation_fr_Text2019), ADR(gc_DbmTranslation_fr_Text2020), ADR(gc_DbmTranslation_fr_Text2021), ADR(gc_DbmTranslation_fr_Text2022), ADR(gc_DbmTranslation_fr_Text2023), ADR(gc_DbmTranslation_fr_Text2024), ADR(gc_DbmTranslation_fr_Text2025), ADR(gc_DbmTranslation_fr_Text2026), ADR(gc_DbmTranslation_fr_Text2027), ADR(gc_DbmTranslation_fr_Text2028), ADR(gc_DbmTranslation_fr_Text2029), ADR(gc_DbmTranslation_fr_Text2030), ADR(gc_DbmTranslation_fr_Text2031), ADR(gc_DbmTranslation_fr_Text2032), ADR(gc_DbmTranslation_fr_Text2033), ADR(gc_DbmTranslation_fr_Text2034), ADR(gc_DbmTranslation_fr_Text2035), ADR(gc_DbmTranslation_fr_Text2036), ADR(gc_DbmTranslation_fr_Text2037), ADR(gc_DbmTranslation_fr_Text2038), ADR(gc_DbmTranslation_fr_Text2039), ADR(gc_DbmTranslation_fr_Text2040), ADR(gc_DbmTranslation_fr_Text2041), ADR(gc_DbmTranslation_fr_Text2042), ADR(gc_DbmTranslation_fr_Text2043), ADR(gc_DbmTranslation_fr_Text2044), ADR(gc_DbmTranslation_fr_Text2045), ADR(gc_DbmTranslation_fr_Text2046), ADR(gc_DbmTranslation_fr_Text2047), ADR(gc_DbmTranslation_fr_Text2048), ADR(gc_DbmTranslation_fr_Text2049), ADR(gc_DbmTranslation_fr_Text2050), ADR(gc_DbmTranslation_fr_Text2051), ADR(gc_DbmTranslation_fr_Text2052), ADR(gc_DbmTranslation_fr_Text2053), ADR(gc_DbmTranslation_fr_Text2054), ADR(gc_DbmTranslation_fr_Text2055), ADR(gc_DbmTranslation_fr_Text2056), ADR(gc_DbmTranslation_fr_Text2057), ADR(gc_DbmTranslation_fr_Text2058), ADR(gc_DbmTranslation_fr_Text2059), ADR(gc_DbmTranslation_fr_Text2060), ADR(gc_DbmTranslation_fr_Text2061), ADR(gc_DbmTranslation_fr_Text2062), ADR(gc_DbmTranslation_fr_Text2063), ADR(gc_DbmTranslation_fr_Text2064), ADR(gc_DbmTranslation_fr_Text2065), ADR(gc_DbmTranslation_fr_Text2066), ADR(gc_DbmTranslation_fr_Text2067), ADR(gc_DbmTranslation_fr_Text2068), ADR(gc_DbmTranslation_fr_Text2069), ADR(gc_DbmTranslation_fr_Text2070), ADR(gc_DbmTranslation_fr_Text2071), ADR(gc_DbmTranslation_fr_Text2072), ADR(gc_DbmTranslation_fr_Text2073), ADR(gc_DbmTranslation_fr_Text2074), ADR(gc_DbmTranslation_fr_Text2075), ADR(gc_DbmTranslation_fr_Text2076), ADR(gc_DbmTranslation_fr_Text2077), ADR(gc_DbmTranslation_fr_Text2078), ADR(gc_DbmTranslation_fr_Text2079), ADR(gc_DbmTranslation_fr_Text2080), ADR(gc_DbmTranslation_fr_Text2081), ADR(gc_DbmTranslation_fr_Text2082), ADR(gc_DbmTranslation_fr_Text2083), ADR(gc_DbmTranslation_fr_Text2084), ADR(gc_DbmTranslation_fr_Text2085), ADR(gc_DbmTranslation_fr_Text2086), ADR(gc_DbmTranslation_fr_Text2087), ADR(gc_DbmTranslation_fr_Text2088), ADR(gc_DbmTranslation_fr_Text2089), ADR(gc_DbmTranslation_fr_Text2090), ADR(gc_DbmTranslation_fr_Text2091), ADR(gc_DbmTranslation_fr_Text2092), ADR(gc_DbmTranslation_fr_Text2093), ADR(gc_DbmTranslation_fr_Text2094), ADR(gc_DbmTranslation_fr_Text2095), ADR(gc_DbmTranslation_fr_Text2096), ADR(gc_DbmTranslation_fr_Text2097), ADR(gc_DbmTranslation_fr_Text2098), ADR(gc_DbmTranslation_fr_Text2099), ADR(gc_DbmTranslation_fr_Text2100), ADR(gc_DbmTranslation_fr_Text2101), ADR(gc_DbmTranslation_fr_Text2102), ADR(gc_DbmTranslation_fr_Text2103), ADR(gc_DbmTranslation_fr_Text2104), ADR(gc_DbmTranslation_fr_Text2105), ADR(gc_DbmTranslation_fr_Text2106), ADR(gc_DbmTranslation_fr_Text2107), ADR(gc_DbmTranslation_fr_Text2108), ADR(gc_DbmTranslation_fr_Text2109), ADR(gc_DbmTranslation_fr_Text2110), ADR(gc_DbmTranslation_fr_Text2111), ADR(gc_DbmTranslation_fr_Text2112), ADR(gc_DbmTranslation_fr_Text2113), ADR(gc_DbmTranslation_fr_Text2114), ADR(gc_DbmTranslation_fr_Text2115), ADR(gc_DbmTranslation_fr_Text2116), ADR(gc_DbmTranslation_fr_Text2117), ADR(gc_DbmTranslation_fr_Text2118), ADR(gc_DbmTranslation_fr_Text2119), ADR(gc_DbmTranslation_fr_Text2120), ADR(gc_DbmTranslation_fr_Text2121), ADR(gc_DbmTranslation_fr_Text2122), ADR(gc_DbmTranslation_fr_Text2123), ADR(gc_DbmTranslation_fr_Text2124), ADR(gc_DbmTranslation_fr_Text2125), ADR(gc_DbmTranslation_fr_Text2126), ADR(gc_DbmTranslation_fr_Text2127), ADR(gc_DbmTranslation_fr_Text2128), ADR(gc_DbmTranslation_fr_Text2129), ADR(gc_DbmTranslation_fr_Text2130), ADR(gc_DbmTranslation_fr_Text2131), ADR(gc_DbmTranslation_fr_Text2132), ADR(gc_DbmTranslation_fr_Text2133), ADR(gc_DbmTranslation_fr_Text2134), ADR(gc_DbmTranslation_fr_Text2135), ADR(gc_DbmTranslation_fr_Text2136), ADR(gc_DbmTranslation_fr_Text2137), ADR(gc_DbmTranslation_fr_Text2138), ADR(gc_DbmTranslation_fr_Text2139), ADR(gc_DbmTranslation_fr_Text2140), ADR(gc_DbmTranslation_fr_Text2141), ADR(gc_DbmTranslation_fr_Text2142), ADR(gc_DbmTranslation_fr_Text2143), ADR(gc_DbmTranslation_fr_Text2144), ADR(gc_DbmTranslation_fr_Text2145), ADR(gc_DbmTranslation_fr_Text2146), ADR(gc_DbmTranslation_fr_Text2147), ADR(gc_DbmTranslation_fr_Text2148), ADR(gc_DbmTranslation_fr_Text2149), ADR(gc_DbmTranslation_fr_Text2150), ADR(gc_DbmTranslation_fr_Text2151), ADR(gc_DbmTranslation_fr_Text2152), ADR(gc_DbmTranslation_fr_Text2153), ADR(gc_DbmTranslation_fr_Text2154), ADR(gc_DbmTranslation_fr_Text2155), ADR(gc_DbmTranslation_fr_Text2156), ADR(gc_DbmTranslation_fr_Text2157), ADR(gc_DbmTranslation_fr_Text2158), ADR(gc_DbmTranslation_fr_Text2159), ADR(gc_DbmTranslation_fr_Text2160), ADR(gc_DbmTranslation_fr_Text2161), ADR(gc_DbmTranslation_fr_Text2162), ADR(gc_DbmTranslation_fr_Text2163), ADR(gc_DbmTranslation_fr_Text2164), ADR(gc_DbmTranslation_fr_Text2165), ADR(gc_DbmTranslation_fr_Text2166), ADR(gc_DbmTranslation_fr_Text2167), ADR(gc_DbmTranslation_fr_Text2168), ADR(gc_DbmTranslation_fr_Text2169), ADR(gc_DbmTranslation_fr_Text2170), ADR(gc_DbmTranslation_fr_Text2171), ADR(gc_DbmTranslation_fr_Text2172), ADR(gc_DbmTranslation_fr_Text2173), ADR(gc_DbmTranslation_fr_Text2174), ADR(gc_DbmTranslation_fr_Text2175), ADR(gc_DbmTranslation_fr_Text2176), ADR(gc_DbmTranslation_fr_Text2177), ADR(gc_DbmTranslation_fr_Text2178), ADR(gc_DbmTranslation_fr_Text2179), ADR(gc_DbmTranslation_fr_Text2180), ADR(gc_DbmTranslation_fr_Text2181), ADR(gc_DbmTranslation_fr_Text2182), ADR(gc_DbmTranslation_fr_Text2183), ADR(gc_DbmTranslation_fr_Text2184), ADR(gc_DbmTranslation_fr_Text2185), ADR(gc_DbmTranslation_fr_Text2186), ADR(gc_DbmTranslation_fr_Text2187), ADR(gc_DbmTranslation_fr_Text2188), ADR(gc_DbmTranslation_fr_Text2189), ADR(gc_DbmTranslation_fr_Text2190), ADR(gc_DbmTranslation_fr_Text2191), ADR(gc_DbmTranslation_fr_Text2192), ADR(gc_DbmTranslation_fr_Text2193), ADR(gc_DbmTranslation_fr_Text2194), ADR(gc_DbmTranslation_fr_Text2195), ADR(gc_DbmTranslation_fr_Text2196), ADR(gc_DbmTranslation_fr_Text2197), ADR(gc_DbmTranslation_fr_Text2198), ADR(gc_DbmTranslation_fr_Text2199), ADR(gc_DbmTranslation_fr_Text2200), ADR(gc_DbmTranslation_fr_Text2201), ADR(gc_DbmTranslation_fr_Text2202), ADR(gc_DbmTranslation_fr_Text2203), ADR(gc_DbmTranslation_fr_Text2204), ADR(gc_DbmTranslation_fr_Text2205), ADR(gc_DbmTranslation_fr_Text2206), ADR(gc_DbmTranslation_fr_Text2207), ADR(gc_DbmTranslation_fr_Text2208), ADR(gc_DbmTranslation_fr_Text2209), ADR(gc_DbmTranslation_fr_Text2210), ADR(gc_DbmTranslation_fr_Text2211), ADR(gc_DbmTranslation_fr_Text2212), ADR(gc_DbmTranslation_fr_Text2213), ADR(gc_DbmTranslation_fr_Text2214), ADR(gc_DbmTranslation_fr_Text2215), ADR(gc_DbmTranslation_fr_Text2216), ADR(gc_DbmTranslation_fr_Text2217), ADR(gc_DbmTranslation_fr_Text2218), ADR(gc_DbmTranslation_fr_Text2219), ADR(gc_DbmTranslation_fr_Text2220), ADR(gc_DbmTranslation_fr_Text2221), ADR(gc_DbmTranslation_fr_Text2222), ADR(gc_DbmTranslation_fr_Text2223), ADR(gc_DbmTranslation_fr_Text2224), ADR(gc_DbmTranslation_fr_Text2225), ADR(gc_DbmTranslation_fr_Text2226), ADR(gc_DbmTranslation_fr_Text2227), ADR(gc_DbmTranslation_fr_Text2228), ADR(gc_DbmTranslation_fr_Text2229), ADR(gc_DbmTranslation_fr_Text2230), ADR(gc_DbmTranslation_fr_Text2231), ADR(gc_DbmTranslation_fr_Text2232), ADR(gc_DbmTranslation_fr_Text2233), ADR(gc_DbmTranslation_fr_Text2234), ADR(gc_DbmTranslation_fr_Text2235), ADR(gc_DbmTranslation_fr_Text2236), ADR(gc_DbmTranslation_fr_Text2237), ADR(gc_DbmTranslation_fr_Text2238), ADR(gc_DbmTranslation_fr_Text2239), ADR(gc_DbmTranslation_fr_Text2240), ADR(gc_DbmTranslation_fr_Text2241), ADR(gc_DbmTranslation_fr_Text2242), ADR(gc_DbmTranslation_fr_Text2243), ADR(gc_DbmTranslation_fr_Text2244), ADR(gc_DbmTranslation_fr_Text2245), ADR(gc_DbmTranslation_fr_Text2246), ADR(gc_DbmTranslation_fr_Text2247), ADR(gc_DbmTranslation_fr_Text2248), ADR(gc_DbmTranslation_fr_Text2249), ADR(gc_DbmTranslation_fr_Text2250), ADR(gc_DbmTranslation_fr_Text2251), ADR(gc_DbmTranslation_fr_Text2252), ADR(gc_DbmTranslation_fr_Text2253), ADR(gc_DbmTranslation_fr_Text2254), ADR(gc_DbmTranslation_fr_Text2255), ADR(gc_DbmTranslation_fr_Text2256), ADR(gc_DbmTranslation_fr_Text2257), ADR(gc_DbmTranslation_fr_Text2258), ADR(gc_DbmTranslation_fr_Text2259), ADR(gc_DbmTranslation_fr_Text2260), ADR(gc_DbmTranslation_fr_Text2261), ADR(gc_DbmTranslation_fr_Text2262), ADR(gc_DbmTranslation_fr_Text2263), ADR(gc_DbmTranslation_fr_Text2264), ADR(gc_DbmTranslation_fr_Text2265), ADR(gc_DbmTranslation_fr_Text2266), ADR(gc_DbmTranslation_fr_Text2267), ADR(gc_DbmTranslation_fr_Text2268), ADR(gc_DbmTranslation_fr_Text2269), ADR(gc_DbmTranslation_fr_Text2270), ADR(gc_DbmTranslation_fr_Text2271), ADR(gc_DbmTranslation_fr_Text2272), ADR(gc_DbmTranslation_fr_Text2273), ADR(gc_DbmTranslation_fr_Text2274), ADR(gc_DbmTranslation_fr_Text2275), ADR(gc_DbmTranslation_fr_Text2276), ADR(gc_DbmTranslation_fr_Text2277), ADR(gc_DbmTranslation_fr_Text2278), ADR(gc_DbmTranslation_fr_Text2279), ADR(gc_DbmTranslation_fr_Text2280), ADR(gc_DbmTranslation_fr_Text2281), ADR(gc_DbmTranslation_fr_Text2282), ADR(gc_DbmTranslation_fr_Text2283), ADR(gc_DbmTranslation_fr_Text2284), ADR(gc_DbmTranslation_fr_Text2285), ADR(gc_DbmTranslation_fr_Text2286), ADR(gc_DbmTranslation_fr_Text2287), ADR(gc_DbmTranslation_fr_Text2288), ADR(gc_DbmTranslation_fr_Text2289), ADR(gc_DbmTranslation_fr_Text2290), ADR(gc_DbmTranslation_fr_Text2291), ADR(gc_DbmTranslation_fr_Text2292), ADR(gc_DbmTranslation_fr_Text2293), ADR(gc_DbmTranslation_fr_Text2294), ADR(gc_DbmTranslation_fr_Text2295), ADR(gc_DbmTranslation_fr_Text2296), ADR(gc_DbmTranslation_fr_Text2297), ADR(gc_DbmTranslation_fr_Text2298), ADR(gc_DbmTranslation_fr_Text2299), ADR(gc_DbmTranslation_fr_Text2300), ADR(gc_DbmTranslation_fr_Text2301), ADR(gc_DbmTranslation_fr_Text2302), ADR(gc_DbmTranslation_fr_Text2303), ADR(gc_DbmTranslation_fr_Text2304), ADR(gc_DbmTranslation_fr_Text2305), ADR(gc_DbmTranslation_fr_Text2306), ADR(gc_DbmTranslation_fr_Text2307), ADR(gc_DbmTranslation_fr_Text2308), ADR(gc_DbmTranslation_fr_Text2309), ADR(gc_DbmTranslation_fr_Text2310), ADR(gc_DbmTranslation_fr_Text2311), ADR(gc_DbmTranslation_fr_Text2312), ADR(gc_DbmTranslation_fr_Text2313), ADR(gc_DbmTranslation_fr_Text2314), ADR(gc_DbmTranslation_fr_Text2315), ADR(gc_DbmTranslation_fr_Text2316), ADR(gc_DbmTranslation_fr_Text2317), ADR(gc_DbmTranslation_fr_Text2318), ADR(gc_DbmTranslation_fr_Text2319), ADR(gc_DbmTranslation_fr_Text2320), ADR(gc_DbmTranslation_fr_Text2321), ADR(gc_DbmTranslation_fr_Text2322), ADR(gc_DbmTranslation_fr_Text2323), ADR(gc_DbmTranslation_fr_Text2324), ADR(gc_DbmTranslation_fr_Text2325), ADR(gc_DbmTranslation_fr_Text2326), ADR(gc_DbmTranslation_fr_Text2327), ADR(gc_DbmTranslation_fr_Text2328), ADR(gc_DbmTranslation_fr_Text2329), ADR(gc_DbmTranslation_fr_Text2330), ADR(gc_DbmTranslation_fr_Text2331), ADR(gc_DbmTranslation_fr_Text2332), ADR(gc_DbmTranslation_fr_Text2333), ADR(gc_DbmTranslation_fr_Text2334), ADR(gc_DbmTranslation_fr_Text2335), ADR(gc_DbmTranslation_fr_Text2336), ADR(gc_DbmTranslation_fr_Text2337), ADR(gc_DbmTranslation_fr_Text2338), ADR(gc_DbmTranslation_fr_Text2339), ADR(gc_DbmTranslation_fr_Text2340), ADR(gc_DbmTranslation_fr_Text2341), ADR(gc_DbmTranslation_fr_Text2342), ADR(gc_DbmTranslation_fr_Text2343), ADR(gc_DbmTranslation_fr_Text2344), ADR(gc_DbmTranslation_fr_Text2345), ADR(gc_DbmTranslation_fr_Text2346), ADR(gc_DbmTranslation_fr_Text2347), ADR(gc_DbmTranslation_fr_Text2348), ADR(gc_DbmTranslation_fr_Text2349), ADR(gc_DbmTranslation_fr_Text2350), ADR(gc_DbmTranslation_fr_Text2351), ADR(gc_DbmTranslation_fr_Text2352), ADR(gc_DbmTranslation_fr_Text2353), ADR(gc_DbmTranslation_fr_Text2354), ADR(gc_DbVarGrpNameTranslation_fr_Text2355), ADR(gc_DbVarGrpNameTranslation_fr_Text2356), ADR(gc_DbVarGrpNameTranslation_fr_Text2357), ADR(gc_DbVarGrpNameTranslation_fr_Text2358), ADR(gc_DbVarGrpNameTranslation_fr_Text2359), ADR(gc_DbVarGrpNameTranslation_fr_Text2360), ADR(gc_DbVarGrpNameTranslation_fr_Text2361), ADR(gc_DbVarGrpNameTranslation_fr_Text2362), ADR(gc_DbVarGrpNameTranslation_fr_Text2363), ADR(gc_DbVarGrpNameTranslation_fr_Text2364), ADR(gc_DbVarGrpNameTranslation_fr_Text2365), ADR(gc_DbVarGrpNameTranslation_fr_Text2366), ADR(gc_DbVarGrpNameTranslation_fr_Text2367), ADR(gc_DbVarGrpNameTranslation_fr_Text2368), ADR(gc_DbVarGrpNameTranslation_fr_Text2369), ADR(gc_DbVarGrpNameTranslation_fr_Text2370), ADR(gc_DbVarGrpNameTranslation_fr_Text2371)];
  gc_DbmTranslation_fr : TTranslation := (IsoCode := 'fr', EnglishName := "french", NativeName := "french", Texts := ADR(gc_DbmTranslation_fr_Texts));
  DBM_TRANSLATION_TEXT_COUNT : INT := 2372;
  g_DbmTranslations : ARRAY[0..2] OF POINTER TO TTranslation := [ADR(gc_DbmTranslation_de), ADR(gc_DbmTranslation_en), ADR(gc_DbmTranslation_fr)];
END_VAR
